// TwinCAT 3 PLC project TC_Robot_Contro_System_Test
// ProgramVersion: 3.1.4020.4
// libraries:
//   Tc2_MC2, * (Beckhoff Automation GmbH)
//   Tc2_Standard, * (Beckhoff Automation GmbH)
//   Tc2_System, * (Beckhoff Automation GmbH)
//   Tc3_Module, * (Beckhoff Automation GmbH)
//   VisuDialogs, * (System)
// project tree:
//   DUTs/Axis/ Axis.TcPOU
//   DUTs/Delay/ Delay.TcPOU (not stored)
//   DUTs/Filter_Current/ E_TcMatSimDataAreaType_1.TcDUT (not stored), FB_Filter_Current_Hexapod_Robot.TcPOU, FB_TcMatSimObject_1.TcPOU (not stored), ST_Filter_Current_Hexapod_Robot_InitData.TcDUT (not stored), ST_Filter_Current_Hexapod_Robot_Input.TcDUT, ST_Filter_Current_Hexapod_Robot_Output.TcDUT (not stored), ST_TcMatSimObjectDataAreaInfo_1.TcDUT (not stored)
//   DUTs/Hexapod_Leg/ Hexapod_Leg.TcPOU (not stored)
//   DUTs/Mapping/ Leg_Control_Mapping_Model.TcPOU (not stored), Leg_Model_Mapping_Control.TcPOU (not stored), Variable_Control_Mapping_Model.TcPOU (not stored), Variable_Model_Mapping_Control.TcPOU (not stored)
//   DUTs/Robot_Simulink/ E_TcMatSimDataAreaType.TcDUT, FB_TcMatSimObject.TcPOU (not stored), FB_Welding_Control_Circle_86s.TcPOU, ST_TcMatSimObjectDataAreaInfo.TcDUT, ST_Welding_Control_Circle_86s_InitData.TcDUT (not stored), ST_Welding_Control_Circle_86s_Input.TcDUT, ST_Welding_Control_Circle_86s_Output.TcDUT
//   / GlobalTextList.TcGTLO (not stored), PlcTask.TcTTO (not stored), Simulink_Test.TcTTO, 视图管理器.TcVMO (not stored)
//   POUs/ MAIN.TcPOU, Simulink_Model_Generator.TcPOU
//   VISUs/ Visu_Home.TcVIS (not stored), Visu_Power.TcVIS, Visu_Reset.TcVIS (not stored), Visu_SimulinkMove.TcVIS (not stored), Visu_Stand.TcVIS (not stored)
// real-time tasks:
//   TASK PlcTask: cycle T#1ms, priority 8, ADS port 350
//   TASK Simulink_Test: cycle T#1ms, priority 10, ADS port 351
// motion (NC):
//   TASK NC-Task 1 SAF: cycle T#1ms, priority 4, ADS port 501
//   TASK NC-Task 1 SVB: cycle T#1ms, priority 6, ADS port 511
//   AXIS Axis 1 (id 1)
//     Velo: SlowManual=10, FastManual=20
//     OtherSettings: AllowMotionCmdToSlave=true
//     encoder EncType=19
//       EncPara: ScaleFactorNumerator=0.000152590218967, MaxCount=#xffffffff
//     drive DrvType=16
//       DrvPara: MaxCount=#xffffffff
//         TimeComp: TaskDelayCycles=1
//     controller CtrType=1
//       CtrPara: PriorControlFactor=1
//         Observer: BandWidth=20
//   AXIS Axis 2 (id 2)
//     Velo: SlowManual=10, FastManual=20
//     OtherSettings: AllowMotionCmdToSlave=true
//     encoder EncType=19
//       EncPara: ScaleFactorNumerator=0.000152590218967, MaxCount=#xffffffff
//     drive DrvType=16
//       DrvPara: MaxCount=#xffffffff
//         TimeComp: TaskDelayCycles=1
//     controller CtrType=1
//       CtrPara: PriorControlFactor=1
//         Observer: BandWidth=20
//   AXIS Axis 3 (id 3)
//     Velo: SlowManual=10, FastManual=20
//     OtherSettings: AllowMotionCmdToSlave=true
//     encoder EncType=19
//       EncPara: ScaleFactorNumerator=0.000152590218967, MaxCount=#xffffffff
//     drive DrvType=16
//       DrvPara: MaxCount=#xffffffff
//         TimeComp: TaskDelayCycles=1
//     controller CtrType=1
//       CtrPara: PriorControlFactor=1
//         Observer: BandWidth=20
//   AXIS Axis 4 (id 4)
//     Velo: SlowManual=10, FastManual=20
//     OtherSettings: AllowMotionCmdToSlave=true
//     encoder EncType=19
//       EncPara: ScaleFactorNumerator=0.000152590218967, MaxCount=#xffffffff
//     drive DrvType=16
//       DrvPara: MaxCount=#xffffffff
//         TimeComp: TaskDelayCycles=1
//     controller CtrType=1
//       CtrPara: PriorControlFactor=1
//         Observer: BandWidth=20
//   AXIS Axis 5 (id 5)
//     Velo: SlowManual=10, FastManual=20
//     OtherSettings: AllowMotionCmdToSlave=true
//     encoder EncType=19
//       EncPara: ScaleFactorNumerator=0.000152590218967, MaxCount=#xffffffff
//     drive DrvType=16
//       DrvPara: MaxCount=#xffffffff
//         TimeComp: TaskDelayCycles=1
//     controller CtrType=1
//       CtrPara: PriorControlFactor=1
//         Observer: BandWidth=20
//   AXIS Axis 6 (id 6)
//     Velo: SlowManual=10, FastManual=20
//     OtherSettings: AllowMotionCmdToSlave=true
//     encoder EncType=19
//       EncPara: ScaleFactorNumerator=0.000152590218967, MaxCount=#xffffffff
//     drive DrvType=16
//       DrvPara: MaxCount=#xffffffff
//         TimeComp: TaskDelayCycles=1
//     controller CtrType=1
//       CtrPara: PriorControlFactor=1
//         Observer: BandWidth=20
//   AXIS Axis 7 (id 7)
//     Velo: SlowManual=10, FastManual=20
//     OtherSettings: AllowMotionCmdToSlave=true
//     encoder EncType=19
//       EncPara: ScaleFactorNumerator=0.000152590218967, MaxCount=#xffffffff
//     drive DrvType=16
//       DrvPara: MaxCount=#xffffffff
//         TimeComp: TaskDelayCycles=1
//     controller CtrType=1
//       CtrPara: PriorControlFactor=1
//         Observer: BandWidth=20
//   AXIS Axis 8 (id 8)
//     Velo: SlowManual=10, FastManual=20
//     OtherSettings: AllowMotionCmdToSlave=true
//     encoder EncType=19
//       EncPara: ScaleFactorNumerator=0.000152590218967, MaxCount=#xffffffff
//     drive DrvType=16
//       DrvPara: MaxCount=#xffffffff
//         TimeComp: TaskDelayCycles=1
//     controller CtrType=1
//       CtrPara: PriorControlFactor=1
//         Observer: BandWidth=20
//   AXIS Axis 9 (id 9)
//     Velo: SlowManual=10, FastManual=20
//     OtherSettings: AllowMotionCmdToSlave=true
//     encoder EncType=19
//       EncPara: ScaleFactorNumerator=0.000152590218967, MaxCount=#xffffffff
//     drive DrvType=16
//       DrvPara: MaxCount=#xffffffff
//         TimeComp: TaskDelayCycles=1
//     controller CtrType=1
//       CtrPara: PriorControlFactor=1
//         Observer: BandWidth=20
//   AXIS Axis 10 (id 10)
//     Velo: SlowManual=10, FastManual=20
//     OtherSettings: AllowMotionCmdToSlave=true
//     encoder EncType=19
//       EncPara: ScaleFactorNumerator=0.000152590218967, MaxCount=#xffffffff
//     drive DrvType=16
//       DrvPara: MaxCount=#xffffffff
//         TimeComp: TaskDelayCycles=1
//     controller CtrType=1
//       CtrPara: PriorControlFactor=1
//         Observer: BandWidth=20
//   AXIS Axis 11 (id 11)
//     Velo: SlowManual=10, FastManual=20
//     OtherSettings: AllowMotionCmdToSlave=true
//     encoder EncType=19
//       EncPara: ScaleFactorNumerator=0.000152590218967, MaxCount=#xffffffff
//     drive DrvType=16
//       DrvPara: MaxCount=#xffffffff
//         TimeComp: TaskDelayCycles=1
//     controller CtrType=1
//       CtrPara: PriorControlFactor=1
//         Observer: BandWidth=20
//   AXIS Axis 12 (id 12)
//     Velo: SlowManual=10, FastManual=20
//     OtherSettings: AllowMotionCmdToSlave=true
//     encoder EncType=19
//       EncPara: ScaleFactorNumerator=0.000152590218967, MaxCount=#xffffffff
//     drive DrvType=16
//       DrvPara: MaxCount=#xffffffff
//         TimeComp: TaskDelayCycles=1
//     controller CtrType=1
//       CtrPara: PriorControlFactor=1
//         Observer: BandWidth=20
//   AXIS Axis 13 (id 13)
//     Velo: SlowManual=10, FastManual=20
//     OtherSettings: AllowMotionCmdToSlave=true
//     encoder EncType=19
//       EncPara: ScaleFactorNumerator=0.000152590218967, MaxCount=#xffffffff
//     drive DrvType=16
//       DrvPara: MaxCount=#xffffffff
//         TimeComp: TaskDelayCycles=1
//     controller CtrType=1
//       CtrPara: PriorControlFactor=1
//         Observer: BandWidth=20
//   AXIS Axis 14 (id 14)
//     Velo: SlowManual=10, FastManual=20
//     OtherSettings: AllowMotionCmdToSlave=true
//     encoder EncType=19
//       EncPara: ScaleFactorNumerator=0.000152590218967, MaxCount=#xffffffff
//     drive DrvType=16
//       DrvPara: MaxCount=#xffffffff
//         TimeComp: TaskDelayCycles=1
//     controller CtrType=1
//       CtrPara: PriorControlFactor=1
//         Observer: BandWidth=20
//   AXIS Axis 15 (id 15)
//     Velo: SlowManual=10, FastManual=20
//     OtherSettings: AllowMotionCmdToSlave=true
//     encoder EncType=19
//       EncPara: ScaleFactorNumerator=0.000152590218967, MaxCount=#xffffffff
//     drive DrvType=16
//       DrvPara: MaxCount=#xffffffff
//         TimeComp: TaskDelayCycles=1
//     controller CtrType=1
//       CtrPara: PriorControlFactor=1
//         Observer: BandWidth=20
//   AXIS Axis 16 (id 16)
//     Velo: SlowManual=10, FastManual=20
//     OtherSettings: AllowMotionCmdToSlave=true
//     encoder EncType=19
//       EncPara: ScaleFactorNumerator=0.000152590218967, MaxCount=#xffffffff
//     drive DrvType=16
//       DrvPara: MaxCount=#xffffffff
//         TimeComp: TaskDelayCycles=1
//     controller CtrType=1
//       CtrPara: PriorControlFactor=1
//         Observer: BandWidth=20
//   AXIS Axis 17 (id 17)
//     Velo: SlowManual=10, FastManual=20
//     OtherSettings: AllowMotionCmdToSlave=true
//     encoder EncType=19
//       EncPara: ScaleFactorNumerator=0.000152590218967, MaxCount=#xffffffff
//     drive DrvType=16
//       DrvPara: MaxCount=#xffffffff
//         TimeComp: TaskDelayCycles=1
//     controller CtrType=1
//       CtrPara: PriorControlFactor=1
//         Observer: BandWidth=20
//   AXIS Axis 18 (id 18)
//     Velo: SlowManual=10, FastManual=20
//     OtherSettings: AllowMotionCmdToSlave=true
//     encoder EncType=19
//       EncPara: ScaleFactorNumerator=0.000152590218967, MaxCount=#xffffffff
//     drive DrvType=16
//       DrvPara: MaxCount=#xffffffff
//         TimeComp: TaskDelayCycles=1
//     controller CtrType=1
//       CtrPara: PriorControlFactor=1
//         Observer: BandWidth=20
// I/O:
//   DEVICE Device 3 (EtherCAT), AmsNetId 5.41.150.106.4.1
//     Drive 1 (Elmo Drive) [Gold EtherCAT GCON Drive Rev:0x000103F6]
//     Drive 2 (Elmo Drive) [Gold EtherCAT GCON Drive Rev:0x000103F6]
//     Drive 3 (Elmo Drive) [Gold EtherCAT GCON Drive Rev:0x000103F6]
//     Drive 4 (Elmo Drive) [Gold EtherCAT GCON Drive Rev:0x000103F6]
//     Drive 5 (Elmo Drive) [Gold EtherCAT GCON Drive Rev:0x000103F6]
//     Drive 6 (Elmo Drive) [Gold EtherCAT GCON Drive Rev:0x000103F6]
//     Drive 7 (Elmo Drive) [Gold EtherCAT GCON Drive Rev:0x000103F6]
//     Drive 8 (Elmo Drive) [Gold EtherCAT GCON Drive Rev:0x000103F6]
//     Drive 9 (Elmo Drive) [Gold EtherCAT GCON Drive Rev:0x000103F6]
//     Drive 10 (Elmo Drive) [Gold EtherCAT GCON Drive Rev:0x000103F6]
//     Drive 11 (Elmo Drive) [Gold EtherCAT GCON Drive Rev:0x000103F6]
//     Drive 12 (Elmo Drive) [Gold EtherCAT GCON Drive Rev:0x000103F6]
//     Drive 13 (Elmo Drive) [Gold EtherCAT GCON Drive Rev:0x000103F6]
//     Drive 14 (Elmo Drive) [Gold EtherCAT GCON Drive Rev:0x000103F6]
//     Drive 15 (Elmo Drive) [Gold EtherCAT GCON Drive Rev:0x000103F6]
//     Drive 16 (Elmo Drive) [Gold EtherCAT GCON Drive Rev:0x000103F6]
//     Drive 17 (Elmo Drive) [Gold EtherCAT GCON Drive Rev:0x000103F6]
//     Drive 18 (Elmo Drive) [Gold EtherCAT GCON Drive Rev:0x000103F6]
// variable links:
//   NC-Task 1 SAF/Axes/Axis 1 <-> Device 3 (EtherCAT)/Drive 1 (Elmo Drive)
//     Drive/Inputs/In/nDcOutputTime <-> InfoData/DcOutputShift
//     Drive/Inputs/In/nState1 <-> Inputs/Status word
//     Drive/Inputs/In/nState2 <-> Inputs/Status word @bit 8
//     Drive/Inputs/In/nState4 @bit 1 <-> WcState/InputToggle
//     Drive/Inputs/In/nState4 <-> WcState/WcState
//     Drive/Outputs/Out/nCtrl1 <-> Outputs/Control word
//     Drive/Outputs/Out/nCtrl2 <-> Outputs/Control word @bit 8
//     Drive/Outputs/Out/nDataOut1 <-> Outputs/Target Position
//     Enc/Inputs/In/nDataIn1 <-> Inputs/Position actual value
//     Enc/Inputs/In/nDcInputTime <-> InfoData/DcInputShift
//     Enc/Inputs/In/nState4 @bit 1 <-> WcState/InputToggle
//     Enc/Inputs/In/nState4 <-> WcState/WcState
//   NC-Task 1 SAF/Axes/Axis 10 <-> Device 3 (EtherCAT)/Drive 10 (Elmo Drive)
//     Drive/Inputs/In/nDcOutputTime <-> InfoData/DcOutputShift
//     Drive/Inputs/In/nState1 <-> Inputs/Status word
//     Drive/Inputs/In/nState2 <-> Inputs/Status word @bit 8
//     Drive/Inputs/In/nState4 @bit 1 <-> WcState/InputToggle
//     Drive/Inputs/In/nState4 <-> WcState/WcState
//     Drive/Outputs/Out/nCtrl1 <-> Outputs/Control word
//     Drive/Outputs/Out/nCtrl2 <-> Outputs/Control word @bit 8
//     Drive/Outputs/Out/nDataOut1 <-> Outputs/Target Position
//     Enc/Inputs/In/nDataIn1 <-> Inputs/Position actual value
//     Enc/Inputs/In/nDcInputTime <-> InfoData/DcInputShift
//     Enc/Inputs/In/nState4 @bit 1 <-> WcState/InputToggle
//     Enc/Inputs/In/nState4 <-> WcState/WcState
//   NC-Task 1 SAF/Axes/Axis 11 <-> Device 3 (EtherCAT)/Drive 11 (Elmo Drive)
//     Drive/Inputs/In/nDcOutputTime <-> InfoData/DcOutputShift
//     Drive/Inputs/In/nState1 <-> Inputs/Status word
//     Drive/Inputs/In/nState2 <-> Inputs/Status word @bit 8
//     Drive/Inputs/In/nState4 @bit 1 <-> WcState/InputToggle
//     Drive/Inputs/In/nState4 <-> WcState/WcState
//     Drive/Outputs/Out/nCtrl1 <-> Outputs/Control word
//     Drive/Outputs/Out/nCtrl2 <-> Outputs/Control word @bit 8
//     Drive/Outputs/Out/nDataOut1 <-> Outputs/Target Position
//     Enc/Inputs/In/nDataIn1 <-> Inputs/Position actual value
//     Enc/Inputs/In/nDcInputTime <-> InfoData/DcInputShift
//     Enc/Inputs/In/nState4 @bit 1 <-> WcState/InputToggle
//     Enc/Inputs/In/nState4 <-> WcState/WcState
//   NC-Task 1 SAF/Axes/Axis 12 <-> Device 3 (EtherCAT)/Drive 12 (Elmo Drive)
//     Drive/Inputs/In/nDcOutputTime <-> InfoData/DcOutputShift
//     Drive/Inputs/In/nState1 <-> Inputs/Status word
//     Drive/Inputs/In/nState2 <-> Inputs/Status word @bit 8
//     Drive/Inputs/In/nState4 @bit 1 <-> WcState/InputToggle
//     Drive/Inputs/In/nState4 <-> WcState/WcState
//     Drive/Outputs/Out/nCtrl1 <-> Outputs/Control word
//     Drive/Outputs/Out/nCtrl2 <-> Outputs/Control word @bit 8
//     Drive/Outputs/Out/nDataOut1 <-> Outputs/Target Position
//     Enc/Inputs/In/nDataIn1 <-> Inputs/Position actual value
//     Enc/Inputs/In/nDcInputTime <-> InfoData/DcInputShift
//     Enc/Inputs/In/nState4 @bit 1 <-> WcState/InputToggle
//     Enc/Inputs/In/nState4 <-> WcState/WcState
//   NC-Task 1 SAF/Axes/Axis 13 <-> Device 3 (EtherCAT)/Drive 13 (Elmo Drive)
//     Drive/Inputs/In/nDcOutputTime <-> InfoData/DcOutputShift
//     Drive/Inputs/In/nState1 <-> Inputs/Status word
//     Drive/Inputs/In/nState2 <-> Inputs/Status word @bit 8
//     Drive/Inputs/In/nState4 @bit 1 <-> WcState/InputToggle
//     Drive/Inputs/In/nState4 <-> WcState/WcState
//     Drive/Outputs/Out/nCtrl1 <-> Outputs/Control word
//     Drive/Outputs/Out/nCtrl2 <-> Outputs/Control word @bit 8
//     Drive/Outputs/Out/nDataOut1 <-> Outputs/Target Position
//     Enc/Inputs/In/nDataIn1 <-> Inputs/Position actual value
//     Enc/Inputs/In/nDcInputTime <-> InfoData/DcInputShift
//     Enc/Inputs/In/nState4 @bit 1 <-> WcState/InputToggle
//     Enc/Inputs/In/nState4 <-> WcState/WcState
//   NC-Task 1 SAF/Axes/Axis 14 <-> Device 3 (EtherCAT)/Drive 14 (Elmo Drive)
//     Drive/Inputs/In/nDcOutputTime <-> InfoData/DcOutputShift
//     Drive/Inputs/In/nState1 <-> Inputs/Status word
//     Drive/Inputs/In/nState2 <-> Inputs/Status word @bit 8
//     Drive/Inputs/In/nState4 @bit 1 <-> WcState/InputToggle
//     Drive/Inputs/In/nState4 <-> WcState/WcState
//     Drive/Outputs/Out/nCtrl1 <-> Outputs/Control word
//     Drive/Outputs/Out/nCtrl2 <-> Outputs/Control word @bit 8
//     Drive/Outputs/Out/nDataOut1 <-> Outputs/Target Position
//     Enc/Inputs/In/nDataIn1 <-> Inputs/Position actual value
//     Enc/Inputs/In/nDcInputTime <-> InfoData/DcInputShift
//     Enc/Inputs/In/nState4 @bit 1 <-> WcState/InputToggle
//     Enc/Inputs/In/nState4 <-> WcState/WcState
//   NC-Task 1 SAF/Axes/Axis 15 <-> Device 3 (EtherCAT)/Drive 15 (Elmo Drive)
//     Drive/Inputs/In/nDcOutputTime <-> InfoData/DcOutputShift
//     Drive/Inputs/In/nState1 <-> Inputs/Status word
//     Drive/Inputs/In/nState2 <-> Inputs/Status word @bit 8
//     Drive/Inputs/In/nState4 @bit 1 <-> WcState/InputToggle
//     Drive/Inputs/In/nState4 <-> WcState/WcState
//     Drive/Outputs/Out/nCtrl1 <-> Outputs/Control word
//     Drive/Outputs/Out/nCtrl2 <-> Outputs/Control word @bit 8
//     Drive/Outputs/Out/nDataOut1 <-> Outputs/Target Position
//     Enc/Inputs/In/nDataIn1 <-> Inputs/Position actual value
//     Enc/Inputs/In/nDcInputTime <-> InfoData/DcInputShift
//     Enc/Inputs/In/nState4 @bit 1 <-> WcState/InputToggle
//     Enc/Inputs/In/nState4 <-> WcState/WcState
//   NC-Task 1 SAF/Axes/Axis 16 <-> Device 3 (EtherCAT)/Drive 16 (Elmo Drive)
//     Drive/Inputs/In/nDcOutputTime <-> InfoData/DcOutputShift
//     Drive/Inputs/In/nState1 <-> Inputs/Status word
//     Drive/Inputs/In/nState2 <-> Inputs/Status word @bit 8
//     Drive/Inputs/In/nState4 @bit 1 <-> WcState/InputToggle
//     Drive/Inputs/In/nState4 <-> WcState/WcState
//     Drive/Outputs/Out/nCtrl1 <-> Outputs/Control word
//     Drive/Outputs/Out/nCtrl2 <-> Outputs/Control word @bit 8
//     Drive/Outputs/Out/nDataOut1 <-> Outputs/Target Position
//     Enc/Inputs/In/nDataIn1 <-> Inputs/Position actual value
//     Enc/Inputs/In/nDcInputTime <-> InfoData/DcInputShift
//     Enc/Inputs/In/nState4 @bit 1 <-> WcState/InputToggle
//     Enc/Inputs/In/nState4 <-> WcState/WcState
//   NC-Task 1 SAF/Axes/Axis 17 <-> Device 3 (EtherCAT)/Drive 17 (Elmo Drive)
//     Drive/Inputs/In/nDcOutputTime <-> InfoData/DcOutputShift
//     Drive/Inputs/In/nState1 <-> Inputs/Status word
//     Drive/Inputs/In/nState2 <-> Inputs/Status word @bit 8
//     Drive/Inputs/In/nState4 @bit 1 <-> WcState/InputToggle
//     Drive/Inputs/In/nState4 <-> WcState/WcState
//     Drive/Outputs/Out/nCtrl1 <-> Outputs/Control word
//     Drive/Outputs/Out/nCtrl2 <-> Outputs/Control word @bit 8
//     Drive/Outputs/Out/nDataOut1 <-> Outputs/Target Position
//     Enc/Inputs/In/nDataIn1 <-> Inputs/Position actual value
//     Enc/Inputs/In/nDcInputTime <-> InfoData/DcInputShift
//     Enc/Inputs/In/nState4 @bit 1 <-> WcState/InputToggle
//     Enc/Inputs/In/nState4 <-> WcState/WcState
//   NC-Task 1 SAF/Axes/Axis 18 <-> Device 3 (EtherCAT)/Drive 18 (Elmo Drive)
//     Drive/Inputs/In/nDcOutputTime <-> InfoData/DcOutputShift
//     Drive/Inputs/In/nState1 <-> Inputs/Status word
//     Drive/Inputs/In/nState2 <-> Inputs/Status word @bit 8
//     Drive/Inputs/In/nState4 @bit 1 <-> WcState/InputToggle
//     Drive/Inputs/In/nState4 <-> WcState/WcState
//     Drive/Outputs/Out/nCtrl1 <-> Outputs/Control word
//     Drive/Outputs/Out/nCtrl2 <-> Outputs/Control word @bit 8
//     Drive/Outputs/Out/nDataOut1 <-> Outputs/Target Position
//     Enc/Inputs/In/nDataIn1 <-> Inputs/Position actual value
//     Enc/Inputs/In/nDcInputTime <-> InfoData/DcInputShift
//     Enc/Inputs/In/nState4 @bit 1 <-> WcState/InputToggle
//     Enc/Inputs/In/nState4 <-> WcState/WcState
//   NC-Task 1 SAF/Axes/Axis 2 <-> Device 3 (EtherCAT)/Drive 2 (Elmo Drive)
//     Drive/Inputs/In/nDcOutputTime <-> InfoData/DcOutputShift
//     Drive/Inputs/In/nState1 <-> Inputs/Status word
//     Drive/Inputs/In/nState2 <-> Inputs/Status word @bit 8
//     Drive/Inputs/In/nState4 @bit 1 <-> WcState/InputToggle
//     Drive/Inputs/In/nState4 <-> WcState/WcState
//     Drive/Outputs/Out/nCtrl1 <-> Outputs/Control word
//     Drive/Outputs/Out/nCtrl2 <-> Outputs/Control word @bit 8
//     Drive/Outputs/Out/nDataOut1 <-> Outputs/Target Position
//     Enc/Inputs/In/nDataIn1 <-> Inputs/Position actual value
//     Enc/Inputs/In/nDcInputTime <-> InfoData/DcInputShift
//     Enc/Inputs/In/nState4 @bit 1 <-> WcState/InputToggle
//     Enc/Inputs/In/nState4 <-> WcState/WcState
//   NC-Task 1 SAF/Axes/Axis 3 <-> Device 3 (EtherCAT)/Drive 3 (Elmo Drive)
//     Drive/Inputs/In/nDcOutputTime <-> InfoData/DcOutputShift
//     Drive/Inputs/In/nState1 <-> Inputs/Status word
//     Drive/Inputs/In/nState2 <-> Inputs/Status word @bit 8
//     Drive/Inputs/In/nState4 @bit 1 <-> WcState/InputToggle
//     Drive/Inputs/In/nState4 <-> WcState/WcState
//     Drive/Outputs/Out/nCtrl1 <-> Outputs/Control word
//     Drive/Outputs/Out/nCtrl2 <-> Outputs/Control word @bit 8
//     Drive/Outputs/Out/nDataOut1 <-> Outputs/Target Position
//     Enc/Inputs/In/nDataIn1 <-> Inputs/Position actual value
//     Enc/Inputs/In/nDcInputTime <-> InfoData/DcInputShift
//     Enc/Inputs/In/nState4 @bit 1 <-> WcState/InputToggle
//     Enc/Inputs/In/nState4 <-> WcState/WcState
//   NC-Task 1 SAF/Axes/Axis 4 <-> Device 3 (EtherCAT)/Drive 4 (Elmo Drive)
//     Drive/Inputs/In/nDcOutputTime <-> InfoData/DcOutputShift
//     Drive/Inputs/In/nState1 <-> Inputs/Status word
//     Drive/Inputs/In/nState2 <-> Inputs/Status word @bit 8
//     Drive/Inputs/In/nState4 @bit 1 <-> WcState/InputToggle
//     Drive/Inputs/In/nState4 <-> WcState/WcState
//     Drive/Outputs/Out/nCtrl1 <-> Outputs/Control word
//     Drive/Outputs/Out/nCtrl2 <-> Outputs/Control word @bit 8
//     Drive/Outputs/Out/nDataOut1 <-> Outputs/Target Position
//     Enc/Inputs/In/nDataIn1 <-> Inputs/Position actual value
//     Enc/Inputs/In/nDcInputTime <-> InfoData/DcInputShift
//     Enc/Inputs/In/nState4 @bit 1 <-> WcState/InputToggle
//     Enc/Inputs/In/nState4 <-> WcState/WcState
//   NC-Task 1 SAF/Axes/Axis 5 <-> Device 3 (EtherCAT)/Drive 5 (Elmo Drive)
//     Drive/Inputs/In/nDcOutputTime <-> InfoData/DcOutputShift
//     Drive/Inputs/In/nState1 <-> Inputs/Status word
//     Drive/Inputs/In/nState2 <-> Inputs/Status word @bit 8
//     Drive/Inputs/In/nState4 @bit 1 <-> WcState/InputToggle
//     Drive/Inputs/In/nState4 <-> WcState/WcState
//     Drive/Outputs/Out/nCtrl1 <-> Outputs/Control word
//     Drive/Outputs/Out/nCtrl2 <-> Outputs/Control word @bit 8
//     Drive/Outputs/Out/nDataOut1 <-> Outputs/Target Position
//     Enc/Inputs/In/nDataIn1 <-> Inputs/Position actual value
//     Enc/Inputs/In/nDcInputTime <-> InfoData/DcInputShift
//     Enc/Inputs/In/nState4 @bit 1 <-> WcState/InputToggle
//     Enc/Inputs/In/nState4 <-> WcState/WcState
//   NC-Task 1 SAF/Axes/Axis 6 <-> Device 3 (EtherCAT)/Drive 6 (Elmo Drive)
//     Drive/Inputs/In/nDcOutputTime <-> InfoData/DcOutputShift
//     Drive/Inputs/In/nState1 <-> Inputs/Status word
//     Drive/Inputs/In/nState2 <-> Inputs/Status word @bit 8
//     Drive/Inputs/In/nState4 @bit 1 <-> WcState/InputToggle
//     Drive/Inputs/In/nState4 <-> WcState/WcState
//     Drive/Outputs/Out/nCtrl1 <-> Outputs/Control word
//     Drive/Outputs/Out/nCtrl2 <-> Outputs/Control word @bit 8
//     Drive/Outputs/Out/nDataOut1 <-> Outputs/Target Position
//     Enc/Inputs/In/nDataIn1 <-> Inputs/Position actual value
//     Enc/Inputs/In/nDcInputTime <-> InfoData/DcInputShift
//     Enc/Inputs/In/nState4 @bit 1 <-> WcState/InputToggle
//     Enc/Inputs/In/nState4 <-> WcState/WcState
//   NC-Task 1 SAF/Axes/Axis 7 <-> Device 3 (EtherCAT)/Drive 7 (Elmo Drive)
//     Drive/Inputs/In/nDcOutputTime <-> InfoData/DcOutputShift
//     Drive/Inputs/In/nState1 <-> Inputs/Status word
//     Drive/Inputs/In/nState2 <-> Inputs/Status word @bit 8
//     Drive/Inputs/In/nState4 @bit 1 <-> WcState/InputToggle
//     Drive/Inputs/In/nState4 <-> WcState/WcState
//     Drive/Outputs/Out/nCtrl1 <-> Outputs/Control word
//     Drive/Outputs/Out/nCtrl2 <-> Outputs/Control word @bit 8
//     Drive/Outputs/Out/nDataOut1 <-> Outputs/Target Position
//     Enc/Inputs/In/nDataIn1 <-> Inputs/Position actual value
//     Enc/Inputs/In/nDcInputTime <-> InfoData/DcInputShift
//     Enc/Inputs/In/nState4 @bit 1 <-> WcState/InputToggle
//     Enc/Inputs/In/nState4 <-> WcState/WcState
//   NC-Task 1 SAF/Axes/Axis 8 <-> Device 3 (EtherCAT)/Drive 8 (Elmo Drive)
//     Drive/Inputs/In/nDcOutputTime <-> InfoData/DcOutputShift
//     Drive/Inputs/In/nState1 <-> Inputs/Status word
//     Drive/Inputs/In/nState2 <-> Inputs/Status word @bit 8
//     Drive/Inputs/In/nState4 @bit 1 <-> WcState/InputToggle
//     Drive/Inputs/In/nState4 <-> WcState/WcState
//     Drive/Outputs/Out/nCtrl1 <-> Outputs/Control word
//     Drive/Outputs/Out/nCtrl2 <-> Outputs/Control word @bit 8
//     Drive/Outputs/Out/nDataOut1 <-> Outputs/Target Position
//     Enc/Inputs/In/nDataIn1 <-> Inputs/Position actual value
//     Enc/Inputs/In/nDcInputTime <-> InfoData/DcInputShift
//     Enc/Inputs/In/nState4 @bit 1 <-> WcState/InputToggle
//     Enc/Inputs/In/nState4 <-> WcState/WcState
//   NC-Task 1 SAF/Axes/Axis 9 <-> Device 3 (EtherCAT)/Drive 9 (Elmo Drive)
//     Drive/Inputs/In/nDcOutputTime <-> InfoData/DcOutputShift
//     Drive/Inputs/In/nState1 <-> Inputs/Status word
//     Drive/Inputs/In/nState2 <-> Inputs/Status word @bit 8
//     Drive/Inputs/In/nState4 @bit 1 <-> WcState/InputToggle
//     Drive/Inputs/In/nState4 <-> WcState/WcState
//     Drive/Outputs/Out/nCtrl1 <-> Outputs/Control word
//     Drive/Outputs/Out/nCtrl2 <-> Outputs/Control word @bit 8
//     Drive/Outputs/Out/nDataOut1 <-> Outputs/Target Position
//     Enc/Inputs/In/nDataIn1 <-> Inputs/Position actual value
//     Enc/Inputs/In/nDcInputTime <-> InfoData/DcInputShift
//     Enc/Inputs/In/nState4 @bit 1 <-> WcState/InputToggle
//     Enc/Inputs/In/nState4 <-> WcState/WcState
//   TC_Robot_Contro_System_Test/TC_Robot_Contro_System_Test Instance <-> Device 3 (EtherCAT)/Drive 1 (Elmo Drive)
//     PlcTask Inputs/MAIN.Current_Turque_Value[1] <-> Inputs_1/Current actual value
//   TC_Robot_Contro_System_Test/TC_Robot_Contro_System_Test Instance <-> Device 3 (EtherCAT)/Drive 10 (Elmo Drive)
//     PlcTask Inputs/MAIN.Current_Turque_Value[10] <-> Inputs_1/Current actual value
//   TC_Robot_Contro_System_Test/TC_Robot_Contro_System_Test Instance <-> Device 3 (EtherCAT)/Drive 11 (Elmo Drive)
//     PlcTask Inputs/MAIN.Current_Turque_Value[11] <-> Inputs_1/Current actual value
//   TC_Robot_Contro_System_Test/TC_Robot_Contro_System_Test Instance <-> Device 3 (EtherCAT)/Drive 12 (Elmo Drive)
//     PlcTask Inputs/MAIN.Current_Turque_Value[12] <-> Inputs_1/Current actual value
//   TC_Robot_Contro_System_Test/TC_Robot_Contro_System_Test Instance <-> Device 3 (EtherCAT)/Drive 13 (Elmo Drive)
//     PlcTask Inputs/MAIN.Current_Turque_Value[13] <-> Inputs_1/Current actual value
//   TC_Robot_Contro_System_Test/TC_Robot_Contro_System_Test Instance <-> Device 3 (EtherCAT)/Drive 14 (Elmo Drive)
//     PlcTask Inputs/MAIN.Current_Turque_Value[14] <-> Inputs_1/Current actual value
//   TC_Robot_Contro_System_Test/TC_Robot_Contro_System_Test Instance <-> Device 3 (EtherCAT)/Drive 15 (Elmo Drive)
//     PlcTask Inputs/MAIN.Current_Turque_Value[15] <-> Inputs_1/Current actual value
//   TC_Robot_Contro_System_Test/TC_Robot_Contro_System_Test Instance <-> Device 3 (EtherCAT)/Drive 16 (Elmo Drive)
//     PlcTask Inputs/MAIN.Current_Turque_Value[16] <-> Inputs_1/Current actual value
//   TC_Robot_Contro_System_Test/TC_Robot_Contro_System_Test Instance <-> Device 3 (EtherCAT)/Drive 17 (Elmo Drive)
//     PlcTask Inputs/MAIN.Current_Turque_Value[17] <-> Inputs_1/Current actual value
//   TC_Robot_Contro_System_Test/TC_Robot_Contro_System_Test Instance <-> Device 3 (EtherCAT)/Drive 18 (Elmo Drive)
//     PlcTask Inputs/MAIN.Current_Turque_Value[18] <-> Inputs_1/Current actual value
//   TC_Robot_Contro_System_Test/TC_Robot_Contro_System_Test Instance <-> Device 3 (EtherCAT)/Drive 2 (Elmo Drive)
//     PlcTask Inputs/MAIN.Current_Turque_Value[2] <-> Inputs_1/Current actual value
//   TC_Robot_Contro_System_Test/TC_Robot_Contro_System_Test Instance <-> Device 3 (EtherCAT)/Drive 3 (Elmo Drive)
//     PlcTask Inputs/MAIN.Current_Turque_Value[3] <-> Inputs_1/Current actual value
//   TC_Robot_Contro_System_Test/TC_Robot_Contro_System_Test Instance <-> Device 3 (EtherCAT)/Drive 4 (Elmo Drive)
//     PlcTask Inputs/MAIN.Current_Turque_Value[4] <-> Inputs_1/Current actual value
//   TC_Robot_Contro_System_Test/TC_Robot_Contro_System_Test Instance <-> Device 3 (EtherCAT)/Drive 5 (Elmo Drive)
//     PlcTask Inputs/MAIN.Current_Turque_Value[5] <-> Inputs_1/Current actual value
//   TC_Robot_Contro_System_Test/TC_Robot_Contro_System_Test Instance <-> Device 3 (EtherCAT)/Drive 6 (Elmo Drive)
//     PlcTask Inputs/MAIN.Current_Turque_Value[6] <-> Inputs_1/Current actual value
//   TC_Robot_Contro_System_Test/TC_Robot_Contro_System_Test Instance <-> Device 3 (EtherCAT)/Drive 7 (Elmo Drive)
//     PlcTask Inputs/MAIN.Current_Turque_Value[7] <-> Inputs_1/Current actual value
//   TC_Robot_Contro_System_Test/TC_Robot_Contro_System_Test Instance <-> Device 3 (EtherCAT)/Drive 8 (Elmo Drive)
//     PlcTask Inputs/MAIN.Current_Turque_Value[8] <-> Inputs_1/Current actual value
//   TC_Robot_Contro_System_Test/TC_Robot_Contro_System_Test Instance <-> Device 3 (EtherCAT)/Drive 9 (Elmo Drive)
//     PlcTask Inputs/MAIN.Current_Turque_Value[9] <-> Inputs_1/Current actual value
//   TC_Robot_Contro_System_Test/TC_Robot_Contro_System_Test Instance <-> NC-Task 1 SAF/Axes/Axis 1
//     PlcTask Inputs/MAIN.Axis_Robot[1].AxisRef.NcToPlc <-> Outputs/ToPlc
//     PlcTask Outputs/MAIN.Axis_Robot[1].AxisRef.PlcToNc <-> Inputs/FromPlc
//   TC_Robot_Contro_System_Test/TC_Robot_Contro_System_Test Instance <-> NC-Task 1 SAF/Axes/Axis 10
//     PlcTask Inputs/MAIN.Axis_Robot[10].AxisRef.NcToPlc <-> Outputs/ToPlc
//     PlcTask Outputs/MAIN.Axis_Robot[10].AxisRef.PlcToNc <-> Inputs/FromPlc
//   TC_Robot_Contro_System_Test/TC_Robot_Contro_System_Test Instance <-> NC-Task 1 SAF/Axes/Axis 11
//     PlcTask Inputs/MAIN.Axis_Robot[11].AxisRef.NcToPlc <-> Outputs/ToPlc
//     PlcTask Outputs/MAIN.Axis_Robot[11].AxisRef.PlcToNc <-> Inputs/FromPlc
//   TC_Robot_Contro_System_Test/TC_Robot_Contro_System_Test Instance <-> NC-Task 1 SAF/Axes/Axis 12
//     PlcTask Inputs/MAIN.Axis_Robot[12].AxisRef.NcToPlc <-> Outputs/ToPlc
//     PlcTask Outputs/MAIN.Axis_Robot[12].AxisRef.PlcToNc <-> Inputs/FromPlc
//   TC_Robot_Contro_System_Test/TC_Robot_Contro_System_Test Instance <-> NC-Task 1 SAF/Axes/Axis 13
//     PlcTask Inputs/MAIN.Axis_Robot[13].AxisRef.NcToPlc <-> Outputs/ToPlc
//     PlcTask Outputs/MAIN.Axis_Robot[13].AxisRef.PlcToNc <-> Inputs/FromPlc
//   TC_Robot_Contro_System_Test/TC_Robot_Contro_System_Test Instance <-> NC-Task 1 SAF/Axes/Axis 14
//     PlcTask Inputs/MAIN.Axis_Robot[14].AxisRef.NcToPlc <-> Outputs/ToPlc
//     PlcTask Outputs/MAIN.Axis_Robot[14].AxisRef.PlcToNc <-> Inputs/FromPlc
//   TC_Robot_Contro_System_Test/TC_Robot_Contro_System_Test Instance <-> NC-Task 1 SAF/Axes/Axis 15
//     PlcTask Inputs/MAIN.Axis_Robot[15].AxisRef.NcToPlc <-> Outputs/ToPlc
//     PlcTask Outputs/MAIN.Axis_Robot[15].AxisRef.PlcToNc <-> Inputs/FromPlc
//   TC_Robot_Contro_System_Test/TC_Robot_Contro_System_Test Instance <-> NC-Task 1 SAF/Axes/Axis 16
//     PlcTask Inputs/MAIN.Axis_Robot[16].AxisRef.NcToPlc <-> Outputs/ToPlc
//     PlcTask Outputs/MAIN.Axis_Robot[16].AxisRef.PlcToNc <-> Inputs/FromPlc
//   TC_Robot_Contro_System_Test/TC_Robot_Contro_System_Test Instance <-> NC-Task 1 SAF/Axes/Axis 17
//     PlcTask Inputs/MAIN.Axis_Robot[17].AxisRef.NcToPlc <-> Outputs/ToPlc
//     PlcTask Outputs/MAIN.Axis_Robot[17].AxisRef.PlcToNc <-> Inputs/FromPlc
//   TC_Robot_Contro_System_Test/TC_Robot_Contro_System_Test Instance <-> NC-Task 1 SAF/Axes/Axis 18
//     PlcTask Inputs/MAIN.Axis_Robot[18].AxisRef.NcToPlc <-> Outputs/ToPlc
//     PlcTask Outputs/MAIN.Axis_Robot[18].AxisRef.PlcToNc <-> Inputs/FromPlc
//   TC_Robot_Contro_System_Test/TC_Robot_Contro_System_Test Instance <-> NC-Task 1 SAF/Axes/Axis 2
//     PlcTask Inputs/MAIN.Axis_Robot[2].AxisRef.NcToPlc <-> Outputs/ToPlc
//     PlcTask Outputs/MAIN.Axis_Robot[2].AxisRef.PlcToNc <-> Inputs/FromPlc
//   TC_Robot_Contro_System_Test/TC_Robot_Contro_System_Test Instance <-> NC-Task 1 SAF/Axes/Axis 3
//     PlcTask Inputs/MAIN.Axis_Robot[3].AxisRef.NcToPlc <-> Outputs/ToPlc
//     PlcTask Outputs/MAIN.Axis_Robot[3].AxisRef.PlcToNc <-> Inputs/FromPlc
//   TC_Robot_Contro_System_Test/TC_Robot_Contro_System_Test Instance <-> NC-Task 1 SAF/Axes/Axis 4
//     PlcTask Inputs/MAIN.Axis_Robot[4].AxisRef.NcToPlc <-> Outputs/ToPlc
//     PlcTask Outputs/MAIN.Axis_Robot[4].AxisRef.PlcToNc <-> Inputs/FromPlc
//   TC_Robot_Contro_System_Test/TC_Robot_Contro_System_Test Instance <-> NC-Task 1 SAF/Axes/Axis 5
//     PlcTask Inputs/MAIN.Axis_Robot[5].AxisRef.NcToPlc <-> Outputs/ToPlc
//     PlcTask Outputs/MAIN.Axis_Robot[5].AxisRef.PlcToNc <-> Inputs/FromPlc
//   TC_Robot_Contro_System_Test/TC_Robot_Contro_System_Test Instance <-> NC-Task 1 SAF/Axes/Axis 6
//     PlcTask Inputs/MAIN.Axis_Robot[6].AxisRef.NcToPlc <-> Outputs/ToPlc
//     PlcTask Outputs/MAIN.Axis_Robot[6].AxisRef.PlcToNc <-> Inputs/FromPlc
//   TC_Robot_Contro_System_Test/TC_Robot_Contro_System_Test Instance <-> NC-Task 1 SAF/Axes/Axis 7
//     PlcTask Inputs/MAIN.Axis_Robot[7].AxisRef.NcToPlc <-> Outputs/ToPlc
//     PlcTask Outputs/MAIN.Axis_Robot[7].AxisRef.PlcToNc <-> Inputs/FromPlc
//   TC_Robot_Contro_System_Test/TC_Robot_Contro_System_Test Instance <-> NC-Task 1 SAF/Axes/Axis 8
//     PlcTask Inputs/MAIN.Axis_Robot[8].AxisRef.NcToPlc <-> Outputs/ToPlc
//     PlcTask Outputs/MAIN.Axis_Robot[8].AxisRef.PlcToNc <-> Inputs/FromPlc
//   TC_Robot_Contro_System_Test/TC_Robot_Contro_System_Test Instance <-> NC-Task 1 SAF/Axes/Axis 9
//     PlcTask Inputs/MAIN.Axis_Robot[9].AxisRef.NcToPlc <-> Outputs/ToPlc
//     PlcTask Outputs/MAIN.Axis_Robot[9].AxisRef.PlcToNc <-> Inputs/FromPlc

CONFIGURATION TC_Robot_Contro_System_Test
    RESOURCE PLC ON TwinCAT3
        TASK Simulink_Test(INTERVAL := T#1ms, PRIORITY := 10);
        PROGRAM Simulink_Model_Generator WITH Simulink_Test : Simulink_Model_Generator;
    END_RESOURCE
END_CONFIGURATION

// ---- DUTs/Filter_Current/ST_Filter_Current_Hexapod_Robot_Input.TcDUT
TYPE ST_Filter_Current_Hexapod_Robot_Input :
STRUCT
	Current_Motor: matrix_18_real_T;
END_STRUCT
END_TYPE

// ---- DUTs/Robot_Simulink/E_TcMatSimDataAreaType.TcDUT
TYPE E_TcMatSimDataAreaType :
(
	NotSpecified := 0,
	Standard,
	InputSrc,
	InputDst,
	OutputSrc,
	OutputDst,
	InternalDa,
	MArea,
	RetainDa
);
END_TYPE

// ---- DUTs/Robot_Simulink/ST_TcMatSimObjectDataAreaInfo.TcDUT
TYPE ST_TcMatSimObjectDataAreaInfo :
STRUCT
	pPlcVar: PVOID;
	pModuleProcImg: PVOID;
	nSize: UDINT;
	nDataAreaId: UDINT;
	eDataAreaType: E_TcMatSimDataAreaType;
END_STRUCT
END_TYPE

// ---- DUTs/Robot_Simulink/ST_Welding_Control_Circle_86s_Input.TcDUT
TYPE ST_Welding_Control_Circle_86s_Input :
STRUCT
	t: LREAL;
END_STRUCT
END_TYPE

// ---- DUTs/Robot_Simulink/ST_Welding_Control_Circle_86s_Output.TcDUT
TYPE ST_Welding_Control_Circle_86s_Output :
STRUCT
	Disp_P: matrix_18_real_T;
END_STRUCT
END_TYPE

// ---- POUs/Simulink_Model_Generator.TcPOU
PROGRAM Simulink_Model_Generator
VAR_INPUT
	
	Axis_Number 		: INT;							// 定义轴数目
	
	ExSetPoint_Execute	: BOOL;							// 机器人外部信号发生使能
	ExtSetPointEnable	: BOOL;							// 外部信号发生信号
	ExtSetPointDisable	: BOOL;							// 外部信号结束信号
	
	T_ALL				: LREAL:=100;						// Simulink模型运动总时长
	t_Interval			: LREAL:=0.001;						// 取样时间间隔，默认为1ms
	t					: LREAL:=0;							// 取样当前时间变量，以0为起点
	
	// ====================Simulink模块相关=====================
	Robot_Simulink		: FB_Welding_Control_Circle_86s(oid:=16#01010020);	// Simulink模型定义
	Mapping_Position	: Variable_Model_Mapping_Control;	// 变量映射			
	
	Filter_Current  	: FB_Filter_Current_Hexapod_Robot(oid:=16#01010030);
	Mapping_Current_Filter	: Variable_Control_Mapping_Model;		// 变量映射	

	
END_VAR
VAR
	Leg_Number			: INT;							// 定义机器人腿数
END_VAR
VAR_OUTPUT
	Model_Position		: ARRAY[1..18] OF LREAL;			// Simulink中各个腿的位置
	ExSetPoint_Position	: ARRAY[1..18] OF LREAL;			// 外部信号位置
	
	Current_Turque_Filter  	: ARRAY[1..18] OF LREAL;		// 滤波后电流
	Current_Turque_Leg		: ARRAY[1..18] OF LREAL;		// Mapping后的电流
	Difference_Position	: ARRAY[1..18] OF LREAL;			// 实际位置与输入位置差值
END_VAR

// =======================子程序使能(永久运行)===================
Variable_Monitor();			// 变量监测子程序使能
Logic_Control();			// 逻辑控制子程序使能
Variable_Set();				// 各动作速度子程序使能

// =======================模型使能=======================
IF ExSetPoint_Execute OR MAIN.Home_Execute THEN
	Robot_Simulink.Execute();	// Simulink模型使能
END_IF

IF MAIN.Power_Execute THEN
	Filter_Current.Execute();
END_IF

// =======================外部信号运动程序=======================
IF ExSetPoint_Execute THEN
	//SetGenerator();			// 使能外部信号发生子程序
	FOR Axis_Number := 1 TO 18 {BY 1} DO
		MAIN.Axis_Robot[Axis_Number].ExtSetPoint(	Drive_ExtSetPointEnable:= ExtSetPointEnable, 
													Drive_ExtSetPointDisable:= ExtSetPointDisable, 
													ExSetPosition:= ExSetPoint_Position[Axis_Number]);
	END_FOR
END_IF


// ======================外部信号发生=========================
IF ExtSetPointEnable THEN	
	t := t + t_Interval;
	ExtSetPointDisable := FALSE;
END_IF

IF t>=T_ALL THEN
	ExtSetPointEnable := FALSE;
	t:=0;
	ExtSetPointDisable := TRUE;
END_IF

ACTION Leg_Action:
// ===================机器人触地信号转换====================
//IF ExtSetPointEnable THEN
//	FOR Leg_Number := 1 TO 6 {BY 1} DO
//		IF Leg_Home_Set[Leg_Number] THEN		// 在可视化中，Leg_Home_Set为点动
//			Axis_Home_Set[1+(Leg_Number-1)*3] := Leg_Home_Set[Leg_Number];
//			Axis_Home_Set[2+(Leg_Number-1)*3] := Leg_Home_Set[Leg_Number];
//			Axis_Home_Set[3+(Leg_Number-1)*3] := Leg_Home_Set[Leg_Number];
//		ELSIF Home_Done[1+(Leg_Number-1)*3] AND Home_Done[2+(Leg_Number-1)*3] AND Home_Done[3+(Leg_Number-1)*3] THEN
//			Leg_Home_Set[Leg_Number] := FALSE; 
//		END_IF
//	END_FOR
//END_IF
END_ACTION

ACTION Logic_Control:
// =====================外部信号发生逻辑========================
IF ExSetPoint_Execute THEN
	MAIN.Home_Execute := FALSE;						// 外部信号发生使能时，机器人调零必须结束
	MAIN.Move_Execute :=0;							// 外部信号发生时，不能进行其他运动
ELSIF NOT ExSetPoint_Execute THEN
	ExtSetPointEnable := 0;						// 外部信号发生不使能时，外部信号不能进入程序
	ExtSetPointDisable :=0;
ELSIF ExtSetPointDisable THEN
	ExtSetPointEnable :=0;						// 外部信号发生停止与外部信号发生开始不能同时进行
END_IF

IF MAIN.Home_Execute OR MAIN.Move_Execute THEN
	ExSetPoint_Execute := FALSE;
END_IF
END_ACTION

ACTION Variable_Monitor:
// ==============实际运动位移和输入位移差值检测区==============
FOR Axis_Number := 1 TO 18 {BY 1} DO
	Difference_Position[Axis_Number] := MAIN.Axis_ActPostion[Axis_Number]- Mapping_Position.Controller_Leg_Variable[Axis_Number]; 
END_FOR

// ===================电流滤波环节===================
FOR Axis_Number := 1 TO 18 {BY 1} DO
	Filter_Current.stInput.Current_Motor[Axis_Number-1] := MAIN.Current_Turque_Value[Axis_Number];
END_FOR	

Current_Turque_Filter := Filter_Current.stOutput.Current_Monitor;
Mapping_Current_Filter(Controller_Leg_Variable:= Current_Turque_Filter, Model_Leg_Variable=> Current_Turque_Leg);
END_ACTION

ACTION Variable_Set:
// ===================外部信号发生电机位置输入值================
FOR Axis_Number := 1 TO 18 {BY 1} DO
	ExSetPoint_Position[Axis_Number]:= Mapping_Position.Controller_Leg_Variable[Axis_Number];
END_FOR

// ===================程序与模型的变量链接===================
Mapping_Position(Model_Leg_Variable:= Model_Position);		// 映射运动学模型中腿编号和控制模型中的电机编号
Robot_Simulink.stInput.t := t;								// 采样时间t与Simulink模型中的采样时间链接
Model_Position := Robot_Simulink.stOutput.Disp_P;			// Simulink中的电机输出位移输入到控制模型
END_ACTION

END_PROGRAM

// ---- DUTs/Robot_Simulink/FB_Welding_Control_Circle_86s.TcPOU
{attribute 'TcDependOnClassFactory' := 'Welding_Control_Circle_86s'}
FUNCTION_BLOCK FB_Welding_Control_Circle_86s EXTENDS FB_TcMatSimObject
VAR_INPUT
	stInput: ST_Welding_Control_Circle_86s_Input;
END_VAR
VAR_OUTPUT
	stOutput: ST_Welding_Control_Circle_86s_Output;
END_VAR
VAR
	stInitData: ST_Welding_Control_Circle_86s_InitData;
	arrDataAreas: ARRAY[1..2] OF ST_TcMatSimObjectDataAreaInfo;
	bParametersVerified: BOOL;
END_VAR

PROPERTY CallBy_Online : TctModuleCallByType
GET
hResult := GetObjPara(16#00000000,sizeof(CallBy_Online),adr(CallBy_Online));
END_GET
SET
hResult := SetObjPara(16#00000000,sizeof(CallBy_Online),adr(CallBy_Online));
END_SET
END_PROPERTY

PROPERTY CallBy_Startup : TctModuleCallByType
GET
CallBy_Startup := stInitData.CallBy;
END_GET
SET
stInitData.CallBy := CallBy_Startup;
END_SET
END_PROPERTY

PROPERTY ContextInfoArr_0_TaskCycleTimeNs_Online : UDINT
GET
hResult := GetObjPara(16#03002080,sizeof(ContextInfoArr_0_TaskCycleTimeNs_Online),adr(ContextInfoArr_0_TaskCycleTimeNs_Online));
END_GET
SET
hResult := SetObjPara(16#03002080,sizeof(ContextInfoArr_0_TaskCycleTimeNs_Online),adr(ContextInfoArr_0_TaskCycleTimeNs_Online));
END_SET
END_PROPERTY

PROPERTY ContextInfoArr_0_TaskCycleTimeNs_Startup : UDINT
GET
ContextInfoArr_0_TaskCycleTimeNs_Startup := stInitData.ContextInfoArr_0_TaskCycleTimeNs;
END_GET
SET
stInitData.ContextInfoArr_0_TaskCycleTimeNs := ContextInfoArr_0_TaskCycleTimeNs_Startup;
END_SET
END_PROPERTY

PROPERTY ContextInfoArr_0_TaskOid_Online : OTCID
GET
hResult := GetObjPara(16#03002060,sizeof(ContextInfoArr_0_TaskOid_Online),adr(ContextInfoArr_0_TaskOid_Online));
END_GET
SET
hResult := SetObjPara(16#03002060,sizeof(ContextInfoArr_0_TaskOid_Online),adr(ContextInfoArr_0_TaskOid_Online));
END_SET
END_PROPERTY

PROPERTY ContextInfoArr_0_TaskOid_Startup : OTCID
GET
ContextInfoArr_0_TaskOid_Startup := stInitData.ContextInfoArr_0_TaskOid;
END_GET
SET
stInitData.ContextInfoArr_0_TaskOid := ContextInfoArr_0_TaskOid_Startup;
END_SET
END_PROPERTY

PROPERTY ContextInfoArr_0_TaskPort_Online : UINT
GET
hResult := GetObjPara(16#03002090,sizeof(ContextInfoArr_0_TaskPort_Online),adr(ContextInfoArr_0_TaskPort_Online));
END_GET
SET
hResult := SetObjPara(16#03002090,sizeof(ContextInfoArr_0_TaskPort_Online),adr(ContextInfoArr_0_TaskPort_Online));
END_SET
END_PROPERTY

PROPERTY ContextInfoArr_0_TaskPort_Startup : UINT
GET
ContextInfoArr_0_TaskPort_Startup := stInitData.ContextInfoArr_0_TaskPort;
END_GET
SET
stInitData.ContextInfoArr_0_TaskPort := ContextInfoArr_0_TaskPort_Startup;
END_SET
END_PROPERTY

PROPERTY ContextInfoArr_0_TaskPriority_Online : UDINT
GET
hResult := GetObjPara(16#03002070,sizeof(ContextInfoArr_0_TaskPriority_Online),adr(ContextInfoArr_0_TaskPriority_Online));
END_GET
SET
hResult := SetObjPara(16#03002070,sizeof(ContextInfoArr_0_TaskPriority_Online),adr(ContextInfoArr_0_TaskPriority_Online));
END_SET
END_PROPERTY

PROPERTY ContextInfoArr_0_TaskPriority_Startup : UDINT
GET
ContextInfoArr_0_TaskPriority_Startup := stInitData.ContextInfoArr_0_TaskPriority;
END_GET
SET
stInitData.ContextInfoArr_0_TaskPriority := ContextInfoArr_0_TaskPriority_Startup;
END_SET
END_PROPERTY

PROPERTY ContextInfoArr_0_TaskSortOrder_Online : UDINT
GET
hResult := GetObjPara(16#030020b0,sizeof(ContextInfoArr_0_TaskSortOrder_Online),adr(ContextInfoArr_0_TaskSortOrder_Online));
END_GET
SET
hResult := SetObjPara(16#030020b0,sizeof(ContextInfoArr_0_TaskSortOrder_Online),adr(ContextInfoArr_0_TaskSortOrder_Online));
END_SET
END_PROPERTY

PROPERTY ContextInfoArr_0_TaskSortOrder_Startup : UDINT
GET
ContextInfoArr_0_TaskSortOrder_Startup := stInitData.ContextInfoArr_0_TaskSortOrder;
END_GET
SET
stInitData.ContextInfoArr_0_TaskSortOrder := ContextInfoArr_0_TaskSortOrder_Startup;
END_SET
END_PROPERTY

PROPERTY CycleUpdateExecuted_Online : BOOL
GET
hResult := GetObjPara(16#00000004,sizeof(CycleUpdateExecuted_Online),adr(CycleUpdateExecuted_Online));
END_GET
SET
hResult := SetObjPara(16#00000004,sizeof(CycleUpdateExecuted_Online),adr(CycleUpdateExecuted_Online));
END_SET
END_PROPERTY

METHOD Execute : HRESULT

IF (SUCCEEDED(hResult)) THEN
  hResult := VerifyParameters();
END_IF

	// update DataArea information
SetDataAreaInfo(ADR(arrDataAreas),2);
	
	// call base method
Execute := SUPER^.Execute();
END_METHOD

PROPERTY ExecuteModelCode_Online : BOOL
GET
hResult := GetObjPara(16#00000008,sizeof(ExecuteModelCode_Online),adr(ExecuteModelCode_Online));
END_GET
SET
hResult := SetObjPara(16#00000008,sizeof(ExecuteModelCode_Online),adr(ExecuteModelCode_Online));
END_SET
END_PROPERTY

PROPERTY ExecuteModelCode_Startup : BOOL
GET
ExecuteModelCode_Startup := stInitData.ExecuteModelCode;
END_GET
SET
stInitData.ExecuteModelCode := ExecuteModelCode_Startup;
END_SET
END_PROPERTY

PROPERTY ExecutionSequence_Online : TctModuleExecutionSequenceType
GET
hResult := GetObjPara(16#00000001,sizeof(ExecutionSequence_Online),adr(ExecutionSequence_Online));
END_GET
SET
hResult := SetObjPara(16#00000001,sizeof(ExecutionSequence_Online),adr(ExecutionSequence_Online));
END_SET
END_PROPERTY

PROPERTY ExecutionSequence_Startup : TctModuleExecutionSequenceType
GET
ExecutionSequence_Startup := stInitData.ExecutionSequence;
END_GET
SET
stInitData.ExecutionSequence := ExecutionSequence_Startup;
END_SET
END_PROPERTY

METHOD FB_init : BOOL
VAR_INPUT
	/// if TRUE, the retain variables are initialized (warm start / cold start)
	bInitRetains: BOOL;
	/// if TRUE, the instance afterwards gets moved into the copy code (online change)
	bInCopyCode: BOOL;
	oid: OTCID;
END_VAR
VAR
	clsId: CLSID;
END_VAR

// initialize flags
bParametersVerified := false;
                    
// set module class id for compatibility check
clsId.Data1 := 16#4f7c9520;
clsId.Data2 := 16#5e7b;
clsId.Data3 := 16#4579;
clsId.Data4[0] := 16#be;
clsId.Data4[1] := 16#6e;
clsId.Data4[2] := 16#10;
clsId.Data4[3] := 16#c0;
clsId.Data4[4] := 16#eb;
clsId.Data4[5] := 16#37;
clsId.Data4[6] := 16#31;
clsId.Data4[7] := 16#6d;

AssignClassId(clsId);
                    
// initialize InitData structure with default values              
stInitData.CallByHdr.indexGroup := 0;
stInitData.CallByHdr.indexOffset := 16#00000000;
stInitData.CallByHdr.cbData := SIZEOF(stInitData.CallBy);
stInitData.CallBy := TctModuleCallByType.Module;
stInitData.ExecutionSequenceHdr.indexGroup := 0;
stInitData.ExecutionSequenceHdr.indexOffset := 16#00000001;
stInitData.ExecutionSequenceHdr.cbData := SIZEOF(stInitData.ExecutionSequence);
stInitData.ExecutionSequence := TctModuleExecutionSequenceType.StateUpdateAfterOutputMapping;
stInitData.StepSizeHdr.indexGroup := 0;
stInitData.StepSizeHdr.indexOffset := 16#00000002;
stInitData.StepSizeHdr.cbData := SIZEOF(stInitData.StepSize);
stInitData.StepSize := TctStepSizeType.UseTaskCycleTime;
stInitData.ExecuteModelCodeHdr.indexGroup := 0;
stInitData.ExecuteModelCodeHdr.indexOffset := 16#00000008;
stInitData.ExecuteModelCodeHdr.cbData := SIZEOF(stInitData.ExecuteModelCode);
stInitData.ExecuteModelCode := 1;
stInitData.ContextInfoArr_0_TaskOidHdr.indexGroup := 0;
stInitData.ContextInfoArr_0_TaskOidHdr.indexOffset := 16#03002060;
stInitData.ContextInfoArr_0_TaskOidHdr.cbData := SIZEOF(stInitData.ContextInfoArr_0_TaskOid);
stInitData.ContextInfoArr_0_TaskPriorityHdr.indexGroup := 0;
stInitData.ContextInfoArr_0_TaskPriorityHdr.indexOffset := 16#03002070;
stInitData.ContextInfoArr_0_TaskPriorityHdr.cbData := SIZEOF(stInitData.ContextInfoArr_0_TaskPriority);
stInitData.ContextInfoArr_0_TaskCycleTimeNsHdr.indexGroup := 0;
stInitData.ContextInfoArr_0_TaskCycleTimeNsHdr.indexOffset := 16#03002080;
stInitData.ContextInfoArr_0_TaskCycleTimeNsHdr.cbData := SIZEOF(stInitData.ContextInfoArr_0_TaskCycleTimeNs);
stInitData.ContextInfoArr_0_TaskPortHdr.indexGroup := 0;
stInitData.ContextInfoArr_0_TaskPortHdr.indexOffset := 16#03002090;
stInitData.ContextInfoArr_0_TaskPortHdr.cbData := SIZEOF(stInitData.ContextInfoArr_0_TaskPort);
stInitData.ContextInfoArr_0_TaskSortOrderHdr.indexGroup := 0;
stInitData.ContextInfoArr_0_TaskSortOrderHdr.indexOffset := 16#030020b0;
stInitData.ContextInfoArr_0_TaskSortOrderHdr.cbData := SIZEOF(stInitData.ContextInfoArr_0_TaskSortOrder);
stInitData.Header.cbData := SIZEOF(stInitData)-SIZEOF(stInitData.Header);
stInitData.Header.uiElmCnt := 9;


// set pointer to InitData structure
SetInitDataInfo(ADR(stInitData));

// set DataArea information
SetDataAreaInfo(ADR(arrDataAreas),2);
arrDataAreas[1].nDataAreaId := 0;
arrDataAreas[1].nSize := SIZEOF(stInput);
arrDataAreas[1].pPlcVar := ADR(stInput);
arrDataAreas[1].pModuleProcImg := 0;
arrDataAreas[1].eDataAreaType := E_TcMatSimDataAreaType.InputDst;
arrDataAreas[2].nDataAreaId := 1;
arrDataAreas[2].nSize := SIZEOF(stOutput);
arrDataAreas[2].pPlcVar := ADR(stOutput);
arrDataAreas[2].pModuleProcImg := 0;
arrDataAreas[2].eDataAreaType := E_TcMatSimDataAreaType.OutputSrc;


// initialize basic interface pointers and return
FB_init := SUCCEEDED(Init(oid));
END_METHOD

PROPERTY InitData : ST_Welding_Control_Circle_86s_InitData
GET
InitData := stInitData;
END_GET
SET
stInitData := InitData;
END_SET
END_PROPERTY

PROPERTY Input_Online : ExtU_output_WeldingDiameter10_T
GET
hResult := GetObjPara(16#80000000,sizeof(Input_Online),adr(Input_Online));
END_GET
SET
hResult := SetObjPara(16#80000000,sizeof(Input_Online),adr(Input_Online));
END_SET
END_PROPERTY

{attribute 'object_name' := 'Internal_SetObjState'}
METHOD PROTECTED Internal_SetObjState
VAR_INPUT
	hr: REFERENCE TO HRESULT;
	nextState: TCOM_STATE;
END_VAR

// update pointer to InitData structure
SetInitDataInfo(ADR(stInitData));
// call base method
SUPER^.Internal_SetObjState(hr,nextState);
END_METHOD

PROPERTY MdlInitialized_Online : BOOL
GET
hResult := GetObjPara(16#00000003,sizeof(MdlInitialized_Online),adr(MdlInitialized_Online));
END_GET
SET
hResult := SetObjPara(16#00000003,sizeof(MdlInitialized_Online),adr(MdlInitialized_Online));
END_SET
END_PROPERTY

PROPERTY ModuleBuildInfo_Online : TctModuleBuildInfoType
GET
hResult := GetObjPara(16#00000007,sizeof(ModuleBuildInfo_Online),adr(ModuleBuildInfo_Online));
END_GET
SET
hResult := SetObjPara(16#00000007,sizeof(ModuleBuildInfo_Online),adr(ModuleBuildInfo_Online));
END_SET
END_PROPERTY

PROPERTY ModuleInfo_Online : TctModuleInfoType
GET
hResult := GetObjPara(16#00000006,sizeof(ModuleInfo_Online),adr(ModuleInfo_Online));
END_GET
SET
hResult := SetObjPara(16#00000006,sizeof(ModuleInfo_Online),adr(ModuleInfo_Online));
END_SET
END_PROPERTY

{attribute 'object_name' := 'SaveOnlineParametersForInit'}
METHOD SaveOnlineParametersForInit : HRESULT
VAR
	idx: UINT;
	pInitElemHdr: POINTER TO TComInitDataElmHdr;
	pData: PVOID;
	nData: UDINT;
END_VAR
VAR CONSTANT
	nInitDataAlignment: UDINT := 4;
END_VAR

// update pointer to InitData structure
SetInitDataInfo(ADR(stInitData));
// call base method
SaveOnlineParametersForInit := SUPER^.SaveOnlineParametersForInit();
END_METHOD

PROPERTY SimulinkTime_Online : LREAL
GET
hResult := GetObjPara(16#00000005,sizeof(SimulinkTime_Online),adr(SimulinkTime_Online));
END_GET
SET
hResult := SetObjPara(16#00000005,sizeof(SimulinkTime_Online),adr(SimulinkTime_Online));
END_SET
END_PROPERTY

PROPERTY StepSize_Online : TctStepSizeType
GET
hResult := GetObjPara(16#00000002,sizeof(StepSize_Online),adr(StepSize_Online));
END_GET
SET
hResult := SetObjPara(16#00000002,sizeof(StepSize_Online),adr(StepSize_Online));
END_SET
END_PROPERTY

PROPERTY StepSize_Startup : TctStepSizeType
GET
StepSize_Startup := stInitData.StepSize;
END_GET
SET
stInitData.StepSize := StepSize_Startup;
END_SET
END_PROPERTY

{attribute 'object_name' := 'VerifyParameters'}
METHOD PRIVATE VerifyParameters : HRESULT
VAR
	moduleCallByParam: TctModuleCallByType;
END_VAR

IF (bParametersVerified) THEN
  VerifyParameters := Tc2_System.E_HRESULTAdsErr.HRESULT_ADS_NOERROR;
ELSE
  VerifyParameters := GetObjPara(stInitData.CallByHdr.indexOffset,SIZEOF(moduleCallByParam),ADR(moduleCallByParam));
  
  // check the "CallBy" parameter to be set to "Module"
  IF (SUCCEEDED(VerifyParameters) AND (moduleCallByParam <> TctModuleCallByType.Module)) THEN
      VerifyParameters := Tc2_System.E_HRESULTAdsErr.INVALIDPARM;
  END_IF
  
  // set the parameters verified flag
  bParametersVerified := SUCCEEDED(VerifyParameters);
END_IF
END_METHOD

END_FUNCTION_BLOCK

// ---- DUTs/Filter_Current/FB_Filter_Current_Hexapod_Robot.TcPOU
{attribute 'TcDependOnClassFactory' := 'Filter_Current_Hexapod_Robot'}
FUNCTION_BLOCK FB_Filter_Current_Hexapod_Robot EXTENDS FB_TcMatSimObject
VAR_INPUT
	stInput: ST_Filter_Current_Hexapod_Robot_Input;
END_VAR
VAR_OUTPUT
	stOutput: ST_Filter_Current_Hexapod_Robot_Output;
END_VAR
VAR
	stInitData: ST_Filter_Current_Hexapod_Robot_InitData;
	arrDataAreas: ARRAY[1..2] OF ST_TcMatSimObjectDataAreaInfo;
	bParametersVerified: BOOL;
END_VAR

PROPERTY CallBy_Online : TctModuleCallByType
GET
hResult := GetObjPara(16#00000000,sizeof(CallBy_Online),adr(CallBy_Online));
END_GET
SET
hResult := SetObjPara(16#00000000,sizeof(CallBy_Online),adr(CallBy_Online));
END_SET
END_PROPERTY

PROPERTY CallBy_Startup : TctModuleCallByType
GET
CallBy_Startup := stInitData.CallBy;
END_GET
SET
stInitData.CallBy := CallBy_Startup;
END_SET
END_PROPERTY

PROPERTY ContextInfoArr_0_TaskCycleTimeNs_Online : UDINT
GET
hResult := GetObjPara(16#03002080,sizeof(ContextInfoArr_0_TaskCycleTimeNs_Online),adr(ContextInfoArr_0_TaskCycleTimeNs_Online));
END_GET
SET
hResult := SetObjPara(16#03002080,sizeof(ContextInfoArr_0_TaskCycleTimeNs_Online),adr(ContextInfoArr_0_TaskCycleTimeNs_Online));
END_SET
END_PROPERTY

PROPERTY ContextInfoArr_0_TaskCycleTimeNs_Startup : UDINT
GET
ContextInfoArr_0_TaskCycleTimeNs_Startup := stInitData.ContextInfoArr_0_TaskCycleTimeNs;
END_GET
SET
stInitData.ContextInfoArr_0_TaskCycleTimeNs := ContextInfoArr_0_TaskCycleTimeNs_Startup;
END_SET
END_PROPERTY

PROPERTY ContextInfoArr_0_TaskOid_Online : OTCID
GET
hResult := GetObjPara(16#03002060,sizeof(ContextInfoArr_0_TaskOid_Online),adr(ContextInfoArr_0_TaskOid_Online));
END_GET
SET
hResult := SetObjPara(16#03002060,sizeof(ContextInfoArr_0_TaskOid_Online),adr(ContextInfoArr_0_TaskOid_Online));
END_SET
END_PROPERTY

PROPERTY ContextInfoArr_0_TaskOid_Startup : OTCID
GET
ContextInfoArr_0_TaskOid_Startup := stInitData.ContextInfoArr_0_TaskOid;
END_GET
SET
stInitData.ContextInfoArr_0_TaskOid := ContextInfoArr_0_TaskOid_Startup;
END_SET
END_PROPERTY

PROPERTY ContextInfoArr_0_TaskPort_Online : UINT
GET
hResult := GetObjPara(16#03002090,sizeof(ContextInfoArr_0_TaskPort_Online),adr(ContextInfoArr_0_TaskPort_Online));
END_GET
SET
hResult := SetObjPara(16#03002090,sizeof(ContextInfoArr_0_TaskPort_Online),adr(ContextInfoArr_0_TaskPort_Online));
END_SET
END_PROPERTY

PROPERTY ContextInfoArr_0_TaskPort_Startup : UINT
GET
ContextInfoArr_0_TaskPort_Startup := stInitData.ContextInfoArr_0_TaskPort;
END_GET
SET
stInitData.ContextInfoArr_0_TaskPort := ContextInfoArr_0_TaskPort_Startup;
END_SET
END_PROPERTY

PROPERTY ContextInfoArr_0_TaskPriority_Online : UDINT
GET
hResult := GetObjPara(16#03002070,sizeof(ContextInfoArr_0_TaskPriority_Online),adr(ContextInfoArr_0_TaskPriority_Online));
END_GET
SET
hResult := SetObjPara(16#03002070,sizeof(ContextInfoArr_0_TaskPriority_Online),adr(ContextInfoArr_0_TaskPriority_Online));
END_SET
END_PROPERTY

PROPERTY ContextInfoArr_0_TaskPriority_Startup : UDINT
GET
ContextInfoArr_0_TaskPriority_Startup := stInitData.ContextInfoArr_0_TaskPriority;
END_GET
SET
stInitData.ContextInfoArr_0_TaskPriority := ContextInfoArr_0_TaskPriority_Startup;
END_SET
END_PROPERTY

PROPERTY ContextInfoArr_0_TaskSortOrder_Online : UDINT
GET
hResult := GetObjPara(16#030020b0,sizeof(ContextInfoArr_0_TaskSortOrder_Online),adr(ContextInfoArr_0_TaskSortOrder_Online));
END_GET
SET
hResult := SetObjPara(16#030020b0,sizeof(ContextInfoArr_0_TaskSortOrder_Online),adr(ContextInfoArr_0_TaskSortOrder_Online));
END_SET
END_PROPERTY

PROPERTY ContextInfoArr_0_TaskSortOrder_Startup : UDINT
GET
ContextInfoArr_0_TaskSortOrder_Startup := stInitData.ContextInfoArr_0_TaskSortOrder;
END_GET
SET
stInitData.ContextInfoArr_0_TaskSortOrder := ContextInfoArr_0_TaskSortOrder_Startup;
END_SET
END_PROPERTY

PROPERTY CycleUpdateExecuted_Online : BOOL
GET
hResult := GetObjPara(16#00000004,sizeof(CycleUpdateExecuted_Online),adr(CycleUpdateExecuted_Online));
END_GET
SET
hResult := SetObjPara(16#00000004,sizeof(CycleUpdateExecuted_Online),adr(CycleUpdateExecuted_Online));
END_SET
END_PROPERTY

METHOD Execute : HRESULT

IF (SUCCEEDED(hResult)) THEN
  hResult := VerifyParameters();
END_IF

	// update DataArea information
SetDataAreaInfo(ADR(arrDataAreas),2);
	
	// call base method
Execute := SUPER^.Execute();
END_METHOD

PROPERTY ExecuteModelCode_Online : BOOL
GET
hResult := GetObjPara(16#00000008,sizeof(ExecuteModelCode_Online),adr(ExecuteModelCode_Online));
END_GET
SET
hResult := SetObjPara(16#00000008,sizeof(ExecuteModelCode_Online),adr(ExecuteModelCode_Online));
END_SET
END_PROPERTY

PROPERTY ExecuteModelCode_Startup : BOOL
GET
ExecuteModelCode_Startup := stInitData.ExecuteModelCode;
END_GET
SET
stInitData.ExecuteModelCode := ExecuteModelCode_Startup;
END_SET
END_PROPERTY

PROPERTY ExecutionSequence_Online : TctModuleExecutionSequenceType
GET
hResult := GetObjPara(16#00000001,sizeof(ExecutionSequence_Online),adr(ExecutionSequence_Online));
END_GET
SET
hResult := SetObjPara(16#00000001,sizeof(ExecutionSequence_Online),adr(ExecutionSequence_Online));
END_SET
END_PROPERTY

PROPERTY ExecutionSequence_Startup : TctModuleExecutionSequenceType
GET
ExecutionSequence_Startup := stInitData.ExecutionSequence;
END_GET
SET
stInitData.ExecutionSequence := ExecutionSequence_Startup;
END_SET
END_PROPERTY

METHOD FB_init : BOOL
VAR_INPUT
	/// if TRUE, the retain variables are initialized (warm start / cold start)
	bInitRetains: BOOL;
	/// if TRUE, the instance afterwards gets moved into the copy code (online change)
	bInCopyCode: BOOL;
	oid: OTCID;
END_VAR
VAR
	clsId: CLSID;
END_VAR

// initialize flags
bParametersVerified := false;
                    
// set module class id for compatibility check
clsId.Data1 := 16#4ef20903;
clsId.Data2 := 16#d648;
clsId.Data3 := 16#49c7;
clsId.Data4[0] := 16#a9;
clsId.Data4[1] := 16#06;
clsId.Data4[2] := 16#8c;
clsId.Data4[3] := 16#fc;
clsId.Data4[4] := 16#20;
clsId.Data4[5] := 16#50;
clsId.Data4[6] := 16#7f;
clsId.Data4[7] := 16#b3;

AssignClassId(clsId);
                    
// initialize InitData structure with default values              
stInitData.CallByHdr.indexGroup := 0;
stInitData.CallByHdr.indexOffset := 16#00000000;
stInitData.CallByHdr.cbData := SIZEOF(stInitData.CallBy);
stInitData.CallBy := TctModuleCallByType.Module;
stInitData.ExecutionSequenceHdr.indexGroup := 0;
stInitData.ExecutionSequenceHdr.indexOffset := 16#00000001;
stInitData.ExecutionSequenceHdr.cbData := SIZEOF(stInitData.ExecutionSequence);
stInitData.ExecutionSequence := TctModuleExecutionSequenceType.StateUpdateAfterOutputMapping;
stInitData.StepSizeHdr.indexGroup := 0;
stInitData.StepSizeHdr.indexOffset := 16#00000002;
stInitData.StepSizeHdr.cbData := SIZEOF(stInitData.StepSize);
stInitData.StepSize := TctStepSizeType.UseTaskCycleTime;
stInitData.ExecuteModelCodeHdr.indexGroup := 0;
stInitData.ExecuteModelCodeHdr.indexOffset := 16#00000008;
stInitData.ExecuteModelCodeHdr.cbData := SIZEOF(stInitData.ExecuteModelCode);
stInitData.ExecuteModelCode := 1;
stInitData.ModelParametersHdr.indexGroup := 0;
stInitData.ModelParametersHdr.indexOffset := 16#83000000;
stInitData.ModelParametersHdr.cbData := SIZEOF(stInitData.ModelParameters);
stInitData.ModelParameters.DiscreteFilter_NumCoef[0] := 1.25663706143591720e+01;
stInitData.ModelParameters.DiscreteFilter_NumCoef[1] := 1.25663706143591720e+01;
stInitData.ModelParameters.DiscreteFilter_DenCoef[0] := 2.01256637061435910e+03;
stInitData.ModelParameters.DiscreteFilter_DenCoef[1] := -1.98743362938564090e+03;
stInitData.ModelParameters.DiscreteFilter_InitialStates := 0.00000000000000000e+00;
stInitData.ModelParameters.DiscreteFilter1_NumCoef[0] := 1.25663706143591720e+01;
stInitData.ModelParameters.DiscreteFilter1_NumCoef[1] := 1.25663706143591720e+01;
stInitData.ModelParameters.DiscreteFilter1_DenCoef[0] := 2.01256637061435910e+03;
stInitData.ModelParameters.DiscreteFilter1_DenCoef[1] := -1.98743362938564090e+03;
stInitData.ModelParameters.DiscreteFilter1_InitialStates := 0.00000000000000000e+00;
stInitData.ModelParameters.DiscreteFilter2_NumCoef[0] := 1.25663706143591720e+01;
stInitData.ModelParameters.DiscreteFilter2_NumCoef[1] := 1.25663706143591720e+01;
stInitData.ModelParameters.DiscreteFilter2_DenCoef[0] := 2.01256637061435910e+03;
stInitData.ModelParameters.DiscreteFilter2_DenCoef[1] := -1.98743362938564090e+03;
stInitData.ModelParameters.DiscreteFilter2_InitialStates := 0.00000000000000000e+00;
stInitData.ModelParameters.DiscreteFilter3_NumCoef[0] := 1.25663706143591720e+01;
stInitData.ModelParameters.DiscreteFilter3_NumCoef[1] := 1.25663706143591720e+01;
stInitData.ModelParameters.DiscreteFilter3_DenCoef[0] := 2.01256637061435910e+03;
stInitData.ModelParameters.DiscreteFilter3_DenCoef[1] := -1.98743362938564090e+03;
stInitData.ModelParameters.DiscreteFilter3_InitialStates := 0.00000000000000000e+00;
stInitData.ModelParameters.DiscreteFilter4_NumCoef[0] := 1.25663706143591720e+01;
stInitData.ModelParameters.DiscreteFilter4_NumCoef[1] := 1.25663706143591720e+01;
stInitData.ModelParameters.DiscreteFilter4_DenCoef[0] := 2.01256637061435910e+03;
stInitData.ModelParameters.DiscreteFilter4_DenCoef[1] := -1.98743362938564090e+03;
stInitData.ModelParameters.DiscreteFilter4_InitialStates := 0.00000000000000000e+00;
stInitData.ModelParameters.DiscreteFilter5_NumCoef[0] := 1.25663706143591720e+01;
stInitData.ModelParameters.DiscreteFilter5_NumCoef[1] := 1.25663706143591720e+01;
stInitData.ModelParameters.DiscreteFilter5_DenCoef[0] := 2.01256637061435910e+03;
stInitData.ModelParameters.DiscreteFilter5_DenCoef[1] := -1.98743362938564090e+03;
stInitData.ModelParameters.DiscreteFilter5_InitialStates := 0.00000000000000000e+00;
stInitData.ModelParameters.DiscreteFilter6_NumCoef[0] := 1.25663706143591720e+01;
stInitData.ModelParameters.DiscreteFilter6_NumCoef[1] := 1.25663706143591720e+01;
stInitData.ModelParameters.DiscreteFilter6_DenCoef[0] := 2.01256637061435910e+03;
stInitData.ModelParameters.DiscreteFilter6_DenCoef[1] := -1.98743362938564090e+03;
stInitData.ModelParameters.DiscreteFilter6_InitialStates := 0.00000000000000000e+00;
stInitData.ModelParameters.DiscreteFilter7_NumCoef[0] := 1.25663706143591720e+01;
stInitData.ModelParameters.DiscreteFilter7_NumCoef[1] := 1.25663706143591720e+01;
stInitData.ModelParameters.DiscreteFilter7_DenCoef[0] := 2.01256637061435910e+03;
stInitData.ModelParameters.DiscreteFilter7_DenCoef[1] := -1.98743362938564090e+03;
stInitData.ModelParameters.DiscreteFilter7_InitialStates := 0.00000000000000000e+00;
stInitData.ModelParameters.DiscreteFilter8_NumCoef[0] := 1.25663706143591720e+01;
stInitData.ModelParameters.DiscreteFilter8_NumCoef[1] := 1.25663706143591720e+01;
stInitData.ModelParameters.DiscreteFilter8_DenCoef[0] := 2.01256637061435910e+03;
stInitData.ModelParameters.DiscreteFilter8_DenCoef[1] := -1.98743362938564090e+03;
stInitData.ModelParameters.DiscreteFilter8_InitialStates := 0.00000000000000000e+00;
stInitData.ModelParameters.DiscreteFilter9_NumCoef[0] := 1.25663706143591720e+01;
stInitData.ModelParameters.DiscreteFilter9_NumCoef[1] := 1.25663706143591720e+01;
stInitData.ModelParameters.DiscreteFilter9_DenCoef[0] := 2.01256637061435910e+03;
stInitData.ModelParameters.DiscreteFilter9_DenCoef[1] := -1.98743362938564090e+03;
stInitData.ModelParameters.DiscreteFilter9_InitialStates := 0.00000000000000000e+00;
stInitData.ModelParameters.DiscreteFilter10_NumCoef[0] := 1.25663706143591720e+01;
stInitData.ModelParameters.DiscreteFilter10_NumCoef[1] := 1.25663706143591720e+01;
stInitData.ModelParameters.DiscreteFilter10_DenCoef[0] := 2.01256637061435910e+03;
stInitData.ModelParameters.DiscreteFilter10_DenCoef[1] := -1.98743362938564090e+03;
stInitData.ModelParameters.DiscreteFilter10_InitialStates := 0.00000000000000000e+00;
stInitData.ModelParameters.DiscreteFilter11_NumCoef[0] := 1.25663706143591720e+01;
stInitData.ModelParameters.DiscreteFilter11_NumCoef[1] := 1.25663706143591720e+01;
stInitData.ModelParameters.DiscreteFilter11_DenCoef[0] := 2.01256637061435910e+03;
stInitData.ModelParameters.DiscreteFilter11_DenCoef[1] := -1.98743362938564090e+03;
stInitData.ModelParameters.DiscreteFilter11_InitialStates := 0.00000000000000000e+00;
stInitData.ModelParameters.DiscreteFilter12_NumCoef[0] := 1.25663706143591720e+01;
stInitData.ModelParameters.DiscreteFilter12_NumCoef[1] := 1.25663706143591720e+01;
stInitData.ModelParameters.DiscreteFilter12_DenCoef[0] := 2.01256637061435910e+03;
stInitData.ModelParameters.DiscreteFilter12_DenCoef[1] := -1.98743362938564090e+03;
stInitData.ModelParameters.DiscreteFilter12_InitialStates := 0.00000000000000000e+00;
stInitData.ModelParameters.DiscreteFilter13_NumCoef[0] := 1.25663706143591720e+01;
stInitData.ModelParameters.DiscreteFilter13_NumCoef[1] := 1.25663706143591720e+01;
stInitData.ModelParameters.DiscreteFilter13_DenCoef[0] := 2.01256637061435910e+03;
stInitData.ModelParameters.DiscreteFilter13_DenCoef[1] := -1.98743362938564090e+03;
stInitData.ModelParameters.DiscreteFilter13_InitialStates := 0.00000000000000000e+00;
stInitData.ModelParameters.DiscreteFilter14_NumCoef[0] := 1.25663706143591720e+01;
stInitData.ModelParameters.DiscreteFilter14_NumCoef[1] := 1.25663706143591720e+01;
stInitData.ModelParameters.DiscreteFilter14_DenCoef[0] := 2.01256637061435910e+03;
stInitData.ModelParameters.DiscreteFilter14_DenCoef[1] := -1.98743362938564090e+03;
stInitData.ModelParameters.DiscreteFilter14_InitialStates := 0.00000000000000000e+00;
stInitData.ModelParameters.DiscreteFilter15_NumCoef[0] := 1.25663706143591720e+01;
stInitData.ModelParameters.DiscreteFilter15_NumCoef[1] := 1.25663706143591720e+01;
stInitData.ModelParameters.DiscreteFilter15_DenCoef[0] := 2.01256637061435910e+03;
stInitData.ModelParameters.DiscreteFilter15_DenCoef[1] := -1.98743362938564090e+03;
stInitData.ModelParameters.DiscreteFilter15_InitialStates := 0.00000000000000000e+00;
stInitData.ModelParameters.DiscreteFilter16_NumCoef[0] := 1.25663706143591720e+01;
stInitData.ModelParameters.DiscreteFilter16_NumCoef[1] := 1.25663706143591720e+01;
stInitData.ModelParameters.DiscreteFilter16_DenCoef[0] := 2.01256637061435910e+03;
stInitData.ModelParameters.DiscreteFilter16_DenCoef[1] := -1.98743362938564090e+03;
stInitData.ModelParameters.DiscreteFilter16_InitialStates := 0.00000000000000000e+00;
stInitData.ModelParameters.DiscreteFilter17_NumCoef[0] := 1.25663706143591720e+01;
stInitData.ModelParameters.DiscreteFilter17_NumCoef[1] := 1.25663706143591720e+01;
stInitData.ModelParameters.DiscreteFilter17_DenCoef[0] := 2.01256637061435910e+03;
stInitData.ModelParameters.DiscreteFilter17_DenCoef[1] := -1.98743362938564090e+03;
stInitData.ModelParameters.DiscreteFilter17_InitialStates := 0.00000000000000000e+00;
stInitData.ContextInfoArr_0_TaskOidHdr.indexGroup := 0;
stInitData.ContextInfoArr_0_TaskOidHdr.indexOffset := 16#03002060;
stInitData.ContextInfoArr_0_TaskOidHdr.cbData := SIZEOF(stInitData.ContextInfoArr_0_TaskOid);
stInitData.ContextInfoArr_0_TaskPriorityHdr.indexGroup := 0;
stInitData.ContextInfoArr_0_TaskPriorityHdr.indexOffset := 16#03002070;
stInitData.ContextInfoArr_0_TaskPriorityHdr.cbData := SIZEOF(stInitData.ContextInfoArr_0_TaskPriority);
stInitData.ContextInfoArr_0_TaskCycleTimeNsHdr.indexGroup := 0;
stInitData.ContextInfoArr_0_TaskCycleTimeNsHdr.indexOffset := 16#03002080;
stInitData.ContextInfoArr_0_TaskCycleTimeNsHdr.cbData := SIZEOF(stInitData.ContextInfoArr_0_TaskCycleTimeNs);
stInitData.ContextInfoArr_0_TaskPortHdr.indexGroup := 0;
stInitData.ContextInfoArr_0_TaskPortHdr.indexOffset := 16#03002090;
stInitData.ContextInfoArr_0_TaskPortHdr.cbData := SIZEOF(stInitData.ContextInfoArr_0_TaskPort);
stInitData.ContextInfoArr_0_TaskSortOrderHdr.indexGroup := 0;
stInitData.ContextInfoArr_0_TaskSortOrderHdr.indexOffset := 16#030020b0;
stInitData.ContextInfoArr_0_TaskSortOrderHdr.cbData := SIZEOF(stInitData.ContextInfoArr_0_TaskSortOrder);
stInitData.Header.cbData := SIZEOF(stInitData)-SIZEOF(stInitData.Header);
stInitData.Header.uiElmCnt := 10;


// set pointer to InitData structure
SetInitDataInfo(ADR(stInitData));

// set DataArea information
SetDataAreaInfo(ADR(arrDataAreas),2);
arrDataAreas[1].nDataAreaId := 0;
arrDataAreas[1].nSize := SIZEOF(stInput);
arrDataAreas[1].pPlcVar := ADR(stInput);
arrDataAreas[1].pModuleProcImg := 0;
arrDataAreas[1].eDataAreaType := E_TcMatSimDataAreaType.InputDst;
arrDataAreas[2].nDataAreaId := 1;
arrDataAreas[2].nSize := SIZEOF(stOutput);
arrDataAreas[2].pPlcVar := ADR(stOutput);
arrDataAreas[2].pModuleProcImg := 0;
arrDataAreas[2].eDataAreaType := E_TcMatSimDataAreaType.OutputSrc;


// initialize basic interface pointers and return
FB_init := SUCCEEDED(Init(oid));
END_METHOD

PROPERTY InitData : ST_Filter_Current_Hexapod_Robot_InitData
GET
InitData := stInitData;
END_GET
SET
stInitData := InitData;
END_SET
END_PROPERTY

PROPERTY Input_Online : ExtU_Filter_Current_Hexapod_R_T
GET
hResult := GetObjPara(16#80000000,sizeof(Input_Online),adr(Input_Online));
END_GET
SET
hResult := SetObjPara(16#80000000,sizeof(Input_Online),adr(Input_Online));
END_SET
END_PROPERTY

{attribute 'object_name' := 'Internal_SetObjState'}
METHOD PROTECTED Internal_SetObjState
VAR_INPUT
	hr: REFERENCE TO HRESULT;
	nextState: TCOM_STATE;
END_VAR

// update pointer to InitData structure
SetInitDataInfo(ADR(stInitData));
// call base method
SUPER^.Internal_SetObjState(hr,nextState);
END_METHOD

PROPERTY MdlInitialized_Online : BOOL
GET
hResult := GetObjPara(16#00000003,sizeof(MdlInitialized_Online),adr(MdlInitialized_Online));
END_GET
SET
hResult := SetObjPara(16#00000003,sizeof(MdlInitialized_Online),adr(MdlInitialized_Online));
END_SET
END_PROPERTY

PROPERTY ModelParameters_Online : P_Filter_Current_Hexapod_Robo_T
GET
hResult := GetObjPara(16#83000000,sizeof(ModelParameters_Online),adr(ModelParameters_Online));
END_GET
SET
hResult := SetObjPara(16#83000000,sizeof(ModelParameters_Online),adr(ModelParameters_Online));
END_SET
END_PROPERTY

PROPERTY ModelParameters_Startup : P_Filter_Current_Hexapod_Robo_T
GET
ModelParameters_Startup := stInitData.ModelParameters;
END_GET
SET
stInitData.ModelParameters := ModelParameters_Startup;
END_SET
END_PROPERTY

PROPERTY ModuleBuildInfo_Online : TctModuleBuildInfoType
GET
hResult := GetObjPara(16#00000007,sizeof(ModuleBuildInfo_Online),adr(ModuleBuildInfo_Online));
END_GET
SET
hResult := SetObjPara(16#00000007,sizeof(ModuleBuildInfo_Online),adr(ModuleBuildInfo_Online));
END_SET
END_PROPERTY

PROPERTY ModuleInfo_Online : TctModuleInfoType
GET
hResult := GetObjPara(16#00000006,sizeof(ModuleInfo_Online),adr(ModuleInfo_Online));
END_GET
SET
hResult := SetObjPara(16#00000006,sizeof(ModuleInfo_Online),adr(ModuleInfo_Online));
END_SET
END_PROPERTY

{attribute 'object_name' := 'SaveOnlineParametersForInit'}
METHOD SaveOnlineParametersForInit : HRESULT
VAR
	idx: UINT;
	pInitElemHdr: POINTER TO TComInitDataElmHdr;
	pData: PVOID;
	nData: UDINT;
END_VAR
VAR CONSTANT
	nInitDataAlignment: UDINT := 4;
END_VAR

// update pointer to InitData structure
SetInitDataInfo(ADR(stInitData));
// call base method
SaveOnlineParametersForInit := SUPER^.SaveOnlineParametersForInit();
END_METHOD

PROPERTY SimulinkTime_Online : LREAL
GET
hResult := GetObjPara(16#00000005,sizeof(SimulinkTime_Online),adr(SimulinkTime_Online));
END_GET
SET
hResult := SetObjPara(16#00000005,sizeof(SimulinkTime_Online),adr(SimulinkTime_Online));
END_SET
END_PROPERTY

PROPERTY StepSize_Online : TctStepSizeType
GET
hResult := GetObjPara(16#00000002,sizeof(StepSize_Online),adr(StepSize_Online));
END_GET
SET
hResult := SetObjPara(16#00000002,sizeof(StepSize_Online),adr(StepSize_Online));
END_SET
END_PROPERTY

PROPERTY StepSize_Startup : TctStepSizeType
GET
StepSize_Startup := stInitData.StepSize;
END_GET
SET
stInitData.StepSize := StepSize_Startup;
END_SET
END_PROPERTY

{attribute 'object_name' := 'VerifyParameters'}
METHOD PRIVATE VerifyParameters : HRESULT
VAR
	moduleCallByParam: TctModuleCallByType;
END_VAR

IF (bParametersVerified) THEN
  VerifyParameters := Tc2_System.E_HRESULTAdsErr.HRESULT_ADS_NOERROR;
ELSE
  VerifyParameters := GetObjPara(stInitData.CallByHdr.indexOffset,SIZEOF(moduleCallByParam),ADR(moduleCallByParam));
  
  // check the "CallBy" parameter to be set to "Module"
  IF (SUCCEEDED(VerifyParameters) AND (moduleCallByParam <> TctModuleCallByType.Module)) THEN
      VerifyParameters := Tc2_System.E_HRESULTAdsErr.INVALIDPARM;
  END_IF
  
  // set the parameters verified flag
  bParametersVerified := SUCCEEDED(VerifyParameters);
END_IF
END_METHOD

END_FUNCTION_BLOCK

// ---- POUs/MAIN.TcPOU
PROGRAM MAIN
VAR_INPUT
	// ===================模块动作信号(按动作先后排列)==========
	Power_Execute 		: BOOL;							// 上电使能控制信号
	Axis_Power			: ARRAY[1..18] OF BOOL;			// 单电机使能
	Robot_Power			: BOOL;							// 机器人所有电机使能
	
	Home_Execute		: BOOL;							// 设置零点程序使能
	//Axis_Start_Back 	: ARRAY[1..18] OF BOOL;			// 单电机找零回退信号
	//Robot_Start_Back	: BOOL;							// 机器人所有电机回退信号
	Leg_Home_Set		: ARRAY[1..6] OF BOOL;	
	Axis_Home_Set		: ARRAY[1..18] OF BOOL;			// 单电机设定零点信号
	Robot_Home_Set		: BOOL;							// 机器人所有电机设定零点信号
	//Home_Set_Position	: ARRAY[1..18] OF LREAL;		// 找到零点后电机到达的位置
	//Delay_On			: ARRAY[1..18] OF BOOL;
	//TON1				: TON;
	
	Move_Execute		: BOOL;							// 绝对运动使能信号
	Robot_Stand_Execute	: BOOL;							// 机器人站立程序使能	
	Axis_Absolute_Eable	: ARRAY[1..18] OF BOOL;			// 单电机绝对运动使能信号
	Robot_Absolute_Eable: ARRAY[1..18] OF BOOL;			// 机器人站立使能信号
	Axis_Move_Position	: ARRAY[1..18] OF LREAL;		// 电机绝对运动位置			
	
	Reset_Execute		: BOOL;							// 电机驱动重置动作发生使能
	Axis_Reset			: ARRAY[1..18] OF BOOL;			// 单电机驱动重置信号使能
	Robot_Reset			: BOOL;							// 机器人整体电机驱动重置
	//Axis_ResetDone		: ARRAY[1..18] OF BOOL;			// 单电机驱动重置完成

END_VAR
VAR
// =======================NC轴变量==========================
	//Leg_Robot			: ARRAY[1..6] OF Hexapod_Leg;	// 定义六足的腿
	Axis_Robot			: ARRAY[1..18] OF Axis;			// 定义六足轴参量(可以调整数据上限来调整电机数目)
	Axis_Delay			: Delay;						// 延迟程序
	Leg_Number			: INT;							// 定义机器人腿数
	Axis_Number 		: INT;							// 定义轴数目
	
	// ===================状态监测变量=======================
	Power_Status	: ARRAY[1..18] OF BOOL;				// 上电监测信号
	Leg_Home_Done	: ARRAY[1..6] OF BOOL;
	Home_Done		: ARRAY[1..18] OF BOOL;				// 找零监测信号
	MoveAbsoluteDone: ARRAY[1..18] OF BOOL;				// 电机运动监测信号
	
	Robot_Error		: BOOL;								// 机器人电机错误信号
	Axis_Error		: ARRAY[1..18] OF BOOL;				// 电机错误监测信号
	Axis_ErrorID	: ARRAY[1..18] OF UDINT;			// 电机错误号码监测信号
	
	Axis_ActPostion	: ARRAY[1..18] OF LREAL;			// 电机轴实际位置
	
	// =======================模块中间变量======================
	//HomeDone_Number	: LREAL :=0;					//完成找零的轴数
	//ExSetPoint_Position	: ARRAY[1..18] OF LREAL;		// 外部信号位置
	//t					: LREAL :=0;
	
	// =======================驱动器信号监测====================
	Current_Turque_Value  AT%IW0 : ARRAY[1..18] OF INT ;//电流、力矩相关值
	Current_Before_Mapping	: ARRAY[1..18] OF LREAL ;	// 将Current_Turque_Value转换数制
	Max_Turque_Value 		: INT ;						// 设置最大力矩边界值
	Mapping_Current			: Variable_Control_Mapping_Model;	// 变量映射	
	Current_After_Mapping	: ARRAY[1..18] OF LREAL;	// 映射后的原始电流值
	
	// ====================Simulink模块相关=====================  
  //Filter_Current  : FB_Filter_Current_Hexapod_Robot(oid:=16#01010030);
  //Current_Turque_Filter  : ARRAY[1..18] OF LREAL;
END_VAR

// =======================子程序使能(永久运行)===================
Variable_Monitor();			// 变量监测子程序使能
Logic_Control();			// 逻辑控制子程序使能
Variable_Set();				// 各动作速度子程序使能
Leg_Action();				// 单腿运动子程序使能
Robot_Action();				// 机器人整体运动子程序使能

// =====================电机驱动重置=============================
IF Reset_Execute THEN
	FOR Axis_Number := 1 TO 18 {BY 1} DO
		Axis_Robot[Axis_Number].Reset(Drive_Reset:= Axis_Reset[Axis_Number]);
	END_FOR
END_IF

// =======================电机上电===============================
IF Power_Execute THEN
	FOR Axis_Number := 1 TO 18 {BY 1} DO
		Axis_Robot[Axis_Number].Power(Axis_Enable:= Axis_Power[Axis_Number]);
	END_FOR
END_IF

// =======================找零程序===============================
IF Home_Execute THEN
	FOR Axis_Number := 1 TO 18 {BY 1} DO
		Axis_Robot[Axis_Number].Home(Drive_Home:= Axis_Home_Set[Axis_Number]);
	END_FOR
END_IF

// =======================站立程序===============================
IF Move_Execute THEN
	FOR Axis_Number := 1 TO 18 {BY 1} DO
		Axis_Robot[Axis_Number].Move_Absolute(	Drive_Move_Absolute:= Axis_Absolute_Eable[Axis_Number], 
												Absolute_Position:= Axis_Move_Position[Axis_Number]);
	END_FOR
END_IF

ACTION Leg_Action:
// ===================机器人单条腿找零程序====================
IF Home_Execute THEN
	FOR Leg_Number := 1 TO 6 {BY 1} DO
		IF Leg_Home_Set[Leg_Number] THEN		// 在可视化中，Leg_Home_Set为点动
			Axis_Home_Set[1+(Leg_Number-1)*3] := Leg_Home_Set[Leg_Number];
			Axis_Home_Set[2+(Leg_Number-1)*3] := Leg_Home_Set[Leg_Number];
			Axis_Home_Set[3+(Leg_Number-1)*3] := Leg_Home_Set[Leg_Number];
		ELSIF Home_Done[1+(Leg_Number-1)*3] AND Home_Done[2+(Leg_Number-1)*3] AND Home_Done[3+(Leg_Number-1)*3] THEN
			Leg_Home_Set[Leg_Number] := FALSE; 
		END_IF
	END_FOR
END_IF
END_ACTION

ACTION Logic_Control:
// =======================控制逻辑区==========================
// 保证所有的动作拥有合理的先后顺序，优化控制逻辑
// 也防止出现两个或两个以上动作同时进行的情况，保证控制安全

// ===================电机驱动重置逻辑========================
//FOR Axis_Number := 1 TO 18 {BY 1} DO
IF Axis_Error[1] OR Axis_Error[2] OR Axis_Error[3] OR Axis_Error[4] OR Axis_Error[5] OR Axis_Error[6]
	 OR Axis_Error[7] OR Axis_Error[8] OR Axis_Error[9] OR Axis_Error[10] OR Axis_Error[11] OR Axis_Error[12]
		OR Axis_Error[13] OR Axis_Error[14] OR Axis_Error[15] OR Axis_Error[16] OR Axis_Error[17] OR Axis_Error[18]
THEN
	Robot_Error := TRUE;
ELSE
	Robot_Error := FALSE;
END_IF
//END_FOR

IF Robot_Error THEN
	Reset_Execute := TRUE;
ELSIF NOT Robot_Error THEN
	Reset_Execute := FALSE;
ELSIF NOT Reset_Execute THEN
	Axis_Reset[Axis_Number] := FALSE;
	Axis_Robot[Axis_Number].Reset(Drive_Reset:= Axis_Reset[Axis_Number]);
END_IF

// =====================上电程序逻辑==========================
IF NOT Power_Execute THEN
	FOR Axis_Number := 1 TO 18 {BY 1} DO
		Axis_Power[Axis_Number] := FALSE;
		Axis_Robot[Axis_Number].Power(Axis_Enable:= Axis_Power[Axis_Number]);
	END_FOR
END_IF

// =====================找零程序逻辑==========================
IF Home_Execute THEN
	FOR Axis_Number := 1 TO 18 {BY 1} DO
		IF Home_Done[Axis_Number] THEN			// 	丝杠到达零点位置后，单电机标零使能位关闭			
			Axis_Home_Set[Axis_Number] :=0;	
			Axis_Robot[Axis_Number].Home(Drive_Home:= Axis_Home_Set[Axis_Number]);
		END_IF
	END_FOR
	Move_Execute :=0;							// 设定零点时，不能进行其他运动
	//ExSetPoint_Execute :=0;
ELSIF NOT Home_Execute THEN
	FOR Axis_Number := 1 TO 18 {BY 1} DO
		//Axis_Start_Back[Axis_Number] :=0;
		Axis_Home_Set[Axis_Number] := 0;
	END_FOR
END_IF

// =====================机器人站立逻辑==========================
IF Move_Execute THEN
	//Absolute_Eable := TRUE;
	Home_Execute := FALSE;						// 站立运动使能时，机器人调零必须结束
	//ExSetPoint_Execute :=0;						// 站立运动时，不能进行其他运动
	FOR Axis_Number := 1 TO 18 {BY 1} DO
		IF MoveAbsoluteDone[Axis_Number] THEN	// 	丝杠到达设定位置后，单电机绝对运动使能位关闭
			Axis_Absolute_Eable[Axis_Number] := FALSE;
		END_IF
	END_FOR
ELSIF NOT Move_Execute THEN						// 站立运动不使能,轴不能运动
	FOR Axis_Number := 1 TO 18 {BY 1} DO
		Axis_Absolute_Eable[Axis_Number] := FALSE;
		Axis_Robot[Axis_Number].Move_Absolute(	Drive_Move_Absolute:= Axis_Absolute_Eable[Axis_Number], 
												Absolute_Position:= Axis_Move_Position[Axis_Number]);
	END_FOR
END_IF
END_ACTION

ACTION Robot_Action:
// =================机器人整体运动命令区======================
// 六足所有电机整体控制

// ====================机器人驱动重置=========================
IF Robot_Reset THEN
	IF Reset_Execute THEN
		Axis_Reset[Axis_Number] := TRUE;
		FOR Axis_Number := 1 TO 18 {BY 1} DO
			Axis_Robot[Axis_Number].Reset(Drive_Reset:= Axis_Reset[Axis_Number]);
		END_FOR
	END_IF
END_IF	

// ===================机器人所有电机上电======================
IF Robot_Power THEN	
	IF Power_Execute THEN
		FOR Axis_Number := 1 TO 18 {BY 1} DO
			Axis_Power[Axis_Number] := TRUE ;
		END_FOR
	END_IF
END_IF
	
// ===================机器人找零程序=======================
IF Robot_Home_Set THEN				// 标零程序
	//Robot_Start_Back := FALSE;
	IF Home_Execute THEN
		Leg_Home_Set[3] := Leg_Home_Set[5] := Leg_Home_Set[1];	// 在整机调零时，1\3\5三条腿同时调零；
		Leg_Home_Set[4] := Leg_Home_Set[6] := Leg_Home_Set[2];	// 在整机调零时，2\4\6三条腿同时调零；
	ELSIF NOT Home_Execute THEN
		FOR Leg_Number := 1 TO 6 {BY 1} DO
			Leg_Home_Set[Leg_Number] := FALSE;
		END_FOR
	END_IF
ELSIF NOT Robot_Home_Set AND NOT Home_Execute THEN
	FOR Axis_Number := 1 TO 18 {BY 1} DO
	Axis_Home_Set[Axis_Number] := FALSE;
	END_FOR
END_IF

// =====================站立程序===============================
IF Robot_Stand_Execute THEN
	IF Move_Execute THEN
		FOR Axis_Number := 1 TO 18 {BY 1} DO
			IF MoveAbsoluteDone[Axis_Number] THEN		// 	丝杠到达设定位置后，单电机绝对运动使能位关闭
				Axis_Absolute_Eable[Axis_Number] := FALSE;
			ELSE
				Axis_Absolute_Eable[Axis_Number] := TRUE;
			END_IF
		END_FOR
	END_IF
ELSIF NOT Robot_Stand_Execute AND NOT Move_Execute THEN 
	FOR Axis_Number := 1 TO 18 {BY 1} DO
		Axis_Absolute_Eable[Axis_Number] := FALSE;
	END_FOR
END_IF
END_ACTION

ACTION Variable_Monitor:
// =====================关键数据信号监测======================

// ==============最大力矩设置区(边界控制条件)=================
FOR Axis_Number := 1 TO 18 {BY 1} DO
	Axis_Robot[Axis_Number].Max_Turque_Value := Max_Turque_Value;
END_FOR

// =======================力矩检测区==========================
FOR Axis_Number := 1 TO 18 {BY 1} DO
	Axis_Robot[Axis_Number].Current_Turque_Value := Current_Turque_Value[Axis_Number];
	Current_Before_Mapping[Axis_Number] := INT_TO_LREAL(Current_Turque_Value[Axis_Number]);
END_FOR
Mapping_Current(Controller_Leg_Variable:= Current_Before_Mapping, Model_Leg_Variable=> Current_After_Mapping);

// ====================轴实际位置检测区=======================
FOR Axis_Number := 1 TO 18 {BY 1} DO
	Axis_ActPostion[Axis_Number] := Axis_Robot[Axis_Number].ActPosition;
END_FOR

// =======================上电状态检测区======================
FOR Axis_Number := 1 TO 18 {BY 1} DO
	Power_Status[Axis_Number] := Axis_Robot[Axis_Number].State_PowerStatus;
END_FOR

// =======================找零状态检测区======================
FOR Axis_Number := 1 TO 18 {BY 1} DO
	Home_Done[Axis_Number] := Axis_Robot[Axis_Number].State_HomeDone;
END_FOR

(*FOR Leg_Number := 1 TO 6 {BY 1} DO
	Leg_Home_Done[Leg_Number] := Leg_Robot[Axis_Number].State_HomeDone;
END_FOR*)

// ===================电机绝对运动状态检测区==================
FOR Axis_Number := 1 TO 18 {BY 1} DO
	MoveAbsoluteDone[Axis_Number] := Axis_Robot[Axis_Number].State_MoveAbsoluteDone;
END_FOR

// =======================电机错误检测区======================
FOR Axis_Number := 1 TO 18 {BY 1} DO
	Axis_Error[Axis_Number] := Axis_Robot[Axis_Number].Axis_Error;
	Axis_ErrorID[Axis_Number] := Axis_Robot[Axis_Number].Axis_ErrorID;
END_FOR
END_ACTION

ACTION Variable_Set:
// =======================速度规定区==========================
FOR Axis_Number := 1 TO 18 {BY 1} DO						//此时每一个电机的速度都是一样的
	Axis_Robot[Axis_Number].Home_Velocity 	:= 20;			//找零速度(Axis_Jog中的速度)
	Axis_Robot[Axis_Number].Move_Relative_Velocity	:=30;	//相对运动速度
END_FOR
IF Home_Execute THEN
	//IF Robot_Home_Set THEN
		Axis_Robot[1].Move_Absolute_Velocity :=17; Axis_Robot[3].Move_Absolute_Velocity :=17; Axis_Robot[4].Move_Absolute_Velocity :=16.74;
		Axis_Robot[6].Move_Absolute_Velocity :=16.74; Axis_Robot[7].Move_Absolute_Velocity :=17.3; Axis_Robot[9].Move_Absolute_Velocity :=17.3;
		Axis_Robot[10].Move_Absolute_Velocity :=16.95; Axis_Robot[12].Move_Absolute_Velocity :=16.95; Axis_Robot[13].Move_Absolute_Velocity :=17;
		Axis_Robot[15].Move_Absolute_Velocity :=17; Axis_Robot[16].Move_Absolute_Velocity :=17; Axis_Robot[18].Move_Absolute_Velocity :=17;
		Axis_Robot[2].Move_Absolute_Velocity :=20; Axis_Robot[5].Move_Absolute_Velocity :=19.8; Axis_Robot[8].Move_Absolute_Velocity :=20;
		Axis_Robot[11].Move_Absolute_Velocity :=20; Axis_Robot[14].Move_Absolute_Velocity :=20; Axis_Robot[17].Move_Absolute_Velocity :=20;
	//ELSIF NOT Robot_Home_Set THEN
		//FOR Axis_Number := 1 TO 18 {BY 1} DO
			//Axis_Robot[Axis_Number].Move_Absolute_Velocity	:=10;
		//END_FOR
	//END_IF
ELSE
	FOR Axis_Number := 1 TO 18 {BY 1} DO
			Axis_Robot[Axis_Number].Move_Absolute_Velocity	:=10;
	END_FOR
END_IF
	

// =======================位置规定区==========================
FOR Axis_Number := 1 TO 18 {BY 1} DO
	Axis_Move_Position[Axis_Number] := 160;
END_FOR

// =====================最大力矩规定区========================
Max_Turque_Value := 1000;

// ============电机设置零点后到达位置规定区(链接到Motor_Position_Generator)================
IF Home_Execute THEN
	FOR Axis_Number := 1 TO 18 {BY 1} DO
		Axis_Robot[Axis_Number].Home_Absolute_Position := Simulink_Model_Generator.Mapping_Position.Controller_Leg_Variable[Axis_Number];
	END_FOR
END_IF

// ===================程序与模型的变量链接===================
//FOR Axis_Number := 1 TO 18 {BY 1} DO
//	Simulink_Model_Generator.Filter_Current.stInput.Current_Motor[Axis_Number-1] := Current_Turque_Value[Axis_Number];
//END_FOR	
//Simulink_Model_Generator.Current_Turque_Filter := Simulink_Model_Generator.Filter_Current.stOutput.Current_Monitor;
END_ACTION

END_PROGRAM

// ---- DUTs/Axis/Axis.TcPOU
FUNCTION_BLOCK Axis
//VAR_INPUT	
//END_VAR
VAR_OUTPUT
	Axis_Error			: BOOL;				// Error signal
	Axis_ErrorID		: UDINT;			// Error ID
	Axis_Moves			: BOOL;				// Status of moving
END_VAR
VAR
	// =============== Done signals MC Block =================
	JogDone			    : BOOL;					// Status of function block MC_Jog
	ResetDone		    : BOOL;					// Status of function block MC_Reset
	HaltDone		    : BOOL;					// Status of function block MC_Halt
	HomeDone		    : BOOL;					// Status of function block MC_Home
  	MoveAbsoluteDone : BOOL;        // Status of function block MC_MoveAbsolute
  	ExtSetPiontDone 	: BOOL;         		// Status of function block MC_ExtSetPointGenDisable

	// =============== Control variables ======================
	//Home_Back_Start	: BOOL;
	//Drive_Home		: BOOL;
	
	// =============== State variables ========================
	Power_StatusEnable	: BOOL;					// Enable feedback
	
	// ============= Velocity, override ,Position==============
	Velocity_Jog		: LREAL;				// Jog velocity
	Velocity_Move		: LREAL;				// Target velocity
	Velocity_Home		: LREAL;				// Home velocity
	Velocity_Absolute	: LREAL;				// MoveAbsolute velocity
	Velocity_Relative	: LREAL;				// MoveRelative velocity
	fOverride 			: LREAL := 100.0;		// Override 100%
  Home_Position   : LREAL;        // The absolute position after Home will be
	
	// =============== Trigger function blocks ================
	
	TriggerHalt	: R_TRIG;				// Trigger to recognize rising edge of halt input
	TriggerReset : R_TRIG;				// Trigger to recognize rising edge of reset input
	
	// =============== Axis reference =========================
	AxisRef			: AXIS_REF;				// Axis reference (process data plc/nc)
	
	// =============== About axis turque ====================
	Axis_Current_Turque 	: INT;
  	Axis_Max_Turque       	: INT;

	// ================= Sensor FeedBack ====================
  	Proximity_Switch      : DINT;
	
	// =============== Motion function blocks =================
	Axis_Power 			: MC_Power;				// FB for enable and override			[上电]
	Axis_Home			: MC_Home;				// FB for axis home						[找零]
	Axis_Reset 			: MC_Reset;				// FB to reset axis						[复位]
	Axis_Jog			: MC_Jog;				// FB to jog axis						[点动]
	Axis_Stop 			: MC_Stop;				// FB to stop axis						[停止]
	Axis_Halt			: MC_Halt;				// FB to halt axis						[停止]
	Axis_Move			: MC_MoveVelocity;		// FB to move axis (velocity movement)	[匀速运动]
	Axis_MoveAbsolute 	: MC_MoveAbsolute;		// FB to move axis absolutely			[绝对位置运动]
	Axis_MoveRelative	: MC_MoveRelative;		// FB to move axis relatively			[相对位置运动]
  	Axis_ActPosition  : MC_ReadActualPosition; // FB to read the actual position of axis  [读取电机轴的实际位置]
	Axis_ActVelocity	: MC_ReadActualVelocity;// FB to read the actual Velocity of axis [读取电机轴的实际速度]
	Axis_Delay			: Delay;				// FB to operate the delay program		[延迟程序]
	Axis_ExtSetPiontEnable	: MC_ExtSetPointGenEnable;	// FB to enable extsetpoint		[外部函数发生使能]
	Axis_ExtSetPiontDisable	: MC_ExtSetPointGenDisable;	// FB to disable extsetpoint	[外部函数结束使能]
  
  // =============== Timer =================
  Delay         : TON;          //[定时器]
END_VAR

PROPERTY ActPosition : LREAL
GET
Axis_ActPosition( Axis:= AxisRef, Enable:= TRUE );
ActPosition := Axis_ActPosition.Position;
END_GET
END_PROPERTY

PROPERTY ActVelocity : LREAL
GET
Axis_ActVelocity( Axis:= AxisRef, Enable:= TRUE,  ActualVelocity=> ActVelocity);
END_GET
END_PROPERTY

PROPERTY Current_Turque_Value : INT
GET
Current_Turque_Value := Axis_Current_Turque;
END_GET
SET
Axis_Current_Turque := Current_Turque_Value;
END_SET
END_PROPERTY

METHOD ExtSetPoint
VAR_INPUT
	Drive_ExtSetPointEnable 	: BOOL;		// 使能外部信号开始信号
	Drive_ExtSetPointDisable 	: BOOL;		// 使能外部信号结束信号
	ExSetPosition				: LREAL;	// 外部信号位置
	//Axis_Current_Turque 		: INT;		// 边界条件：丝杠位置到达两端卡死
END_VAR
// =======================外部信号发生程序==========================

IF NOT Axis_ExtSetPiontEnable.Error THEN
	Axis_ExtSetPiontEnable(	Axis:= AxisRef, 
							Execute:= Drive_ExtSetPointEnable, 
							Position:= ExSetPosition, 
							PositionType:= POSITIONTYPE_ABSOLUTE );
END_IF

IF Axis_ExtSetPiontEnable.Done THEN
	ExtSetPiontDone := 1;
	MC_ExtSetPointGenFeed(	Position:= ExSetPosition, 
							Velocity:= 10, 
							Acceleration:= 10, 
							Direction:= 1, 		// 1 = positive direction
							Axis:= AxisRef );
END_IF	

IF NOT Axis_ExtSetPiontDisable.Error THEN 
	Axis_ExtSetPiontDisable(	Axis:= AxisRef, 
								Execute:= Drive_ExtSetPointDisable);
END_IF
								
IF Axis_ExtSetPiontEnable.Error OR Axis_ExtSetPiontDisable.Error OR ABS(Axis_Current_Turque) > Axis_Max_Turque THEN
	IF Axis_ExtSetPiontEnable.Error OR Axis_ExtSetPiontDisable.Error THEN
		Axis_Error		:= TRUE;
		Axis_ErrorID 	:= Axis_Home.ErrorID;
	END_IF
	Axis_ExtSetPiontEnable(	Axis:= AxisRef, 
							Execute:= 0 );
	Axis_ExtSetPiontDisable(	Axis:= AxisRef, 
								Execute:= 1);
END_IF
END_METHOD

METHOD Halt : BOOL
VAR_INPUT
	DriveHalt		: BOOL;					// Request stop
END_VAR
// =======================电机运动停止程序==========================

IF DriveHalt THEN
	// Move Execute FALSE
	Axis_Move(	Execute	:= FALSE,
				Axis 	:= AxisRef);
ELSE
	// Reset done signal
	HaltDone := FALSE;
END_IF

// Trigger
TriggerHalt(CLK := DriveHalt);

IF TriggerHalt.Q THEN
	Axis_Halt(	Execute	:= TRUE,
				Axis 	:= AxisRef);
ELSE
	Axis_Halt(Axis := AxisRef);
END_IF

// Done / Error / Command aborted
IF Axis_Halt.Done OR Axis_Halt.Error OR Axis_Halt.CommandAborted THEN
	Axis_Error		:= Axis_Halt.Error;
	Axis_ErrorID 	:= Axis_Halt.ErrorID;
	HaltDone 		:= Axis_Halt.Done;
	
	Axis_Move(	Execute	:= FALSE,
				Axis 	:= AxisRef);
				
	Axis_Halt(	Execute	:= FALSE,
				Axis 	:= AxisRef);
END_IF

// =========================================================
END_METHOD

METHOD Home
VAR_INPUT
	//Back_Start 				: BOOL;
	//Velocity_Home	:LREAL;
	//Axis_Current_Turque 	: INT;
	Drive_Home				: BOOL;
END_VAR

VAR
	//HomeSet					: BOOL;
	BackDone				: BOOL;					// 电机退回到顶点位，该标志位使能
END_VAR
// =======================找零程序==========================
// 找零程序过程为：先让丝杠回退，到达机械限位后停止,并用程序将该位置置为零位

//======================丝杠回退========================
Jog_Backward(Drive_Jog_Backward:= (Drive_Home AND (NOT BackDone)));
Jog_Velocity := Velocity_Home;
HomeDone := Axis_MoveAbsolute.Done;					// 找零结束的标志为丝杠伸长到制定距离
	
IF NOT Axis_Home.Error THEN
	IF ABS(Axis_Current_Turque) > Axis_Max_Turque AND NOT BackDone THEN
		//Drive_Home :=0;
		Jog_Backward(Drive_Jog_Backward:= 0);
		Delay(IN:= NOT Delay.Q, PT:=T#200MS, Q=> , ET=> );
		Axis_Home( 	Axis:= AxisRef, 
					Execute:= Delay.Q, 
					Position:= 0, 
					HomingMode:= MC_Direct);
		BackDone := Axis_Home.Done;				
	END_IF
	IF BackDone AND Drive_Home THEN
		Move_Absolute(Drive_Move_Absolute:= TRUE, Absolute_Position:= Home_Position );
		IF Axis_MoveAbsolute.Done THEN
			BackDone := FALSE;
			Drive_Home	:= FALSE;
		END_IF
	END_IF
END_IF

(*IF HomeSet THEN
	Jog_Backward(Drive_Jog_Backward:= 0,  Axis_Current_Turque:= Axis_Current_Turque);
	HomeDone := 1;
END_IF*)

IF Axis_Home.Error OR Axis_Home.CommandAborted OR ABS(Axis_Current_Turque) < Axis_Max_Turque THEN
	IF Axis_Jog.Error THEN
		Axis_Error		:= TRUE;
		Axis_ErrorID 	:= Axis_Home.ErrorID;
	END_IF
	Axis_Home( 	Axis:= AxisRef, 
				Execute:= FALSE);
END_IF

// =========================================================
END_METHOD

PROPERTY Home_Absolute_Position : LREAL
GET
Home_Absolute_Position := Home_Position;
END_GET
SET
Home_Position := Home_Absolute_Position;
END_SET
END_PROPERTY

METHOD Home_Sensor
VAR_INPUT
	Drive_Home				: BOOL;			// 调零使能信号
	Home_Switch				: BOOL;			// 零位调零传感器信号
	//MaxPosition_Swicth		: BOOL;
END_VAR

VAR
	//HomeSet				: BOOL;
	BackDone				: BOOL;					// 电机退回到顶点位，该标志位使能
END_VAR
// =======================找零程序==========================
// 找零程序过程为：先让丝杠回退，当传感器检测到金属表面并反馈信号后, 程序将该位置置为零位

//======================丝杠回退========================
Jog_Backward(Drive_Jog_Backward:= Drive_Home);
Jog_Velocity := Velocity_Home;
HomeDone := Axis_MoveAbsolute.Done;					// 回到零点的标志为丝杠伸长到制定距离
	
IF NOT Axis_Home.Error THEN
	IF Home_Switch AND NOT HomeDone THEN
		Drive_Home :=0;
		Jog_Backward(Drive_Jog_Backward:= Drive_Home);
		Delay(IN:= NOT Delay.Q, PT:=T#200MS, Q=> , ET=> );
		Axis_Home( 	Axis:= AxisRef, 
					Execute:= Delay.Q,
					Position:= 0, 
					HomingMode:= MC_Direct);
		BackDone := Axis_Home.Done;
	END_IF
	IF BackDone THEN
		Move_Absolute(Drive_Move_Absolute:= TRUE, Absolute_Position:= 20);
		IF Axis_MoveAbsolute.Done THEN
			BackDone := FALSE;
		END_IF
	END_IF
END_IF

(*IF HomeSet THEN
	Jog_Backward(Drive_Jog_Backward:= 0,  Axis_Current_Turque:= Axis_Current_Turque);
	HomeDone := 1;
END_IF*)

IF Axis_Home.Error OR Axis_Home.CommandAborted OR ABS(Axis_Current_Turque) < Axis_Max_Turque THEN
	IF Axis_Jog.Error THEN
		Axis_Error		:= TRUE;
		Axis_ErrorID 	:= Axis_Home.ErrorID;
	END_IF
	Axis_Home( 	Axis:= AxisRef, 
				Execute:= FALSE);
END_IF

// =========================================================
END_METHOD

PROPERTY Home_Velocity : LREAL
GET
Home_Velocity := Velocity_Home;
END_GET
SET
Velocity_Home := Home_Velocity;
END_SET
END_PROPERTY

METHOD Jog_Backward
VAR_INPUT
	Drive_Jog_Backward	: BOOL;				//点动后退使能信号
	//Velocity_Jog		: LREAL;			//点动速度
	//Axis_Current_Turque : INT;				//边界条件：丝杠位置到达两端卡死
END_VAR
// =======================点动后退==========================
// 点动后退用在找零中的位置移动

IF NOT Axis_Jog.Error THEN
	Axis_Jog( 	Axis:= AxisRef, 
				JogForward:= 0, 
				JogBackwards:= Drive_Jog_Backward, 
				Mode:= MC_JOGMODE_CONTINOUS, 
				Velocity:= Velocity_Jog);
END_IF

IF Axis_Jog.Error OR Axis_Jog.CommandAborted OR ABS(Axis_Current_Turque) > Axis_Max_Turque THEN
	IF Axis_Jog.Error THEN
		Axis_Error		:= TRUE;
		Axis_ErrorID 	:= Axis_Jog.ErrorID;
	END_IF
	
	Axis_Jog(	JogForward:= 0, 
				JogBackwards:= 0, 
				Axis := AxisRef);
END_IF

(*IF ABS(Axis_Current_Turque) <1000 AND JogDone =1 THEN
	Axis_Jog(	JogForward:= 0, 
				JogBackwards:= 0, 
				Axis := AxisRef);
	JogDone :=0;
END_IF*)
				
// =========================================================
END_METHOD

METHOD Jog_Forward : BOOL
VAR_INPUT
	Drive_Jog_Forward	: BOOL;				//点动前进使能信号
	//Velocity_Jog		: LREAL;			//点动速度
	//Axis_Current_Turque : INT;				//边界条件：丝杠位置到达两端卡死
END_VAR
// =======================点动前进==========================


IF NOT Axis_Jog.Error THEN
	Axis_Jog( 	Axis:= AxisRef, 
				JogForward:= Drive_Jog_Forward, 
				JogBackwards:= 0, 
				Mode:= MC_JOGMODE_CONTINOUS, 
				Velocity:= Velocity_Jog);
END_IF

IF Axis_Jog.Error OR Axis_Jog.CommandAborted OR ABS(Axis_Current_Turque) > Axis_Max_Turque THEN
	IF Axis_Jog.Error THEN
		Axis_Error		:= TRUE;
		Axis_ErrorID 	:= Axis_Jog.ErrorID;
	END_IF
	
	Axis_Jog(	JogForward:= 0, 
				JogBackwards:= 0, 
				Axis := AxisRef);
END_IF

(*IF ABS(Axis_Current_Turque) <1000 AND JogDone =1 THEN
	Axis_Jog(	JogForward:= 0, 
				JogBackwards:= 0, 
				Axis := AxisRef);
	JogDone :=0;
END_IF*)
				
// =========================================================
END_METHOD

// =======================读写点动程序中的速度值==========================

PROPERTY Jog_Velocity : LREAL
GET
Jog_Velocity := Velocity_Jog;
END_GET
SET
Velocity_Jog := Jog_Velocity;
END_SET
END_PROPERTY

PROPERTY Max_Turque_Value : INT
SET
Axis_Max_Turque := Max_Turque_Value;
END_SET
END_PROPERTY

METHOD Move_Absolute
VAR_INPUT
	Drive_Move_Absolute : BOOL;				// 运动使能信号
	Absolute_Position	: LREAL;			// 绝对运动位置
	//Move_Velocity		: LREAL;			// 运动速度
	//Axis_Current_Turque : INT;			// 边界条件：丝杠位置到达两端卡死
END_VAR
// =======================绝对运动==========================

IF NOT Axis_MoveAbsolute.Error THEN
	Axis_MoveAbsolute(	Axis:= AxisRef, 
						Execute:= Drive_Move_Absolute, 
						Position:= Absolute_Position, 
						Velocity:= Velocity_Absolute, 
						BufferMode:= MC_Aborting );
	MoveAbsoluteDone := Axis_MoveAbsolute.Done;			// 运动到指定位置后置位
END_IF

IF Axis_MoveAbsolute.Error OR Axis_MoveAbsolute.CommandAborted OR ABS(Axis_Current_Turque) > Axis_Max_Turque THEN
	IF Axis_MoveAbsolute.Error THEN
		Axis_Error		:= TRUE;
		Axis_ErrorID 	:= Axis_MoveAbsolute.ErrorID;
	END_IF
	
	Axis_MoveAbsolute(	Axis:= AxisRef, 
						Execute:= 0, 
						BufferMode:= MC_Aborting);
END_IF

// =========================================================
END_METHOD

// =======================读写绝对运动程序中的速度值==========================

PROPERTY Move_Absolute_Velocity : LREAL
GET
Move_Absolute_Velocity := Velocity_Absolute;
END_GET
SET
Velocity_Absolute := Move_Absolute_Velocity;
END_SET
END_PROPERTY

METHOD Move_Backward
VAR_INPUT
	Move_Backward_Start : BOOL;					//匀速后退使能信号
	//Axis_Current_Turque : INT;					//边界条件：丝杠位置到达两端卡死
END_VAR
// =======================匀速后退==========================

// Not error
IF NOT Axis_Move.Error THEN
	Axis_Move(	Execute 	:= Move_Backward_Start,
				Velocity 	:= Velocity_Move,
				Direction 	:= MC_Negative_Direction,
				Axis 		:= AxisRef );
END_IF

// Error / Command aborted
IF Axis_Move.Error OR Axis_Move.CommandAborted OR ABS(Axis_Current_Turque) > Axis_Max_Turque THEN
	IF Axis_Move.Error THEN
		Axis_Error		:= TRUE;
		Axis_ErrorID 	:= Axis_Move.ErrorID;
	END_IF
	
	Axis_Move(	Execute	:= FALSE,
				Axis 	:= AxisRef);
END_IF

// =========================================================
END_METHOD

METHOD Move_Fordward
VAR_INPUT
	Move_Forward_Start : BOOL;					//匀速前进使能信号
	//Axis_Current_Turque : INT;					//边界条件：丝杠位置到达两端卡死
END_VAR
// =======================匀速前进==========================

// Not error
IF NOT Axis_Move.Error THEN
	Axis_Move(	Execute 	:= Move_Forward_Start,
				Velocity 	:= Velocity_Move,
				Direction 	:= MC_Positive_Direction,
				Axis 		:= AxisRef );
END_IF

// Error / Command aborted
IF Axis_Move.Error OR Axis_Move.CommandAborted OR ABS(Axis_Current_Turque) > Axis_Max_Turque THEN
	IF Axis_Move.Error THEN
		Axis_Error		:= TRUE;
		Axis_ErrorID 	:= Axis_Move.ErrorID;
	END_IF
	
	Axis_Move(	Execute	:= FALSE,
				Axis 	:= AxisRef);
END_IF

// =========================================================
END_METHOD

METHOD Move_Relative
VAR_INPUT
	Drive_Move_Relative		: BOOL;				// 运动使能信号
	Relative_Position		: LREAL;			// 相对运动位置
	//Move_Velocity			: LREAL;			// 运动速度
	//Axis_Current_Turque 	: INT;				// 边界条件：丝杠位置到达两端卡死
END_VAR
// =======================相对运动==========================

IF NOT Axis_MoveRelative.Error THEN
	Axis_MoveRelative(	Axis:= AxisRef, 
						Execute:= Drive_Move_Relative, 
						Distance:= Relative_Position, 
						Velocity:= Velocity_Relative, 
						BufferMode:= MC_Aborting );
END_IF

IF Axis_MoveRelative.Error OR Axis_MoveRelative.CommandAborted OR ABS(Axis_Current_Turque) > Axis_Max_Turque THEN
	IF Axis_MoveRelative.Error THEN
		Axis_Error		:= TRUE;
		Axis_ErrorID 	:= Axis_MoveRelative.ErrorID;
	END_IF
	
	Axis_MoveRelative(	Axis:= AxisRef, 
						Execute:= 0, 
						BufferMode:= MC_Aborting);
END_IF

// =========================================================
END_METHOD

// =======================读写相对运动程序中的速度值==========================

PROPERTY Move_Relative_Velocity : LREAL
GET
Move_Relative_Velocity := Velocity_Relative;
END_GET
SET
Velocity_Relative := Move_Relative_Velocity;
END_SET
END_PROPERTY

PROPERTY Move_Velocity : LREAL
GET
Move_Velocity := Velocity_Move;
END_GET
SET
Velocity_Move :=Move_Velocity :=10;
END_SET
END_PROPERTY

METHOD Power
VAR_INPUT
	Axis_Enable : BOOL;
END_VAR
// =======================上电程序==========================

Axis_Power(	Enable 			:= Axis_Enable, 
			Enable_Positive	:= Axis_Enable, 
			Enable_Negative	:= Axis_Enable, 
			Override		:= fOverride,
			Axis			:= AxisRef,
			Status			=> Power_StatusEnable);
			
IF Axis_Power.Error THEN
	Axis_Error		:= TRUE;
	Axis_ErrorID 	:= Axis_Power.ErrorID;
END_IF

AxisRef.ReadStatus();

Axis_Moves := AxisRef.Status.Moving;

// ==========================================================
END_METHOD

METHOD Reset
VAR_INPUT
	Drive_Reset		: BOOL;					// Request reset
END_VAR
// =====================驱动重置程序==========================

IF NOT Drive_Reset THEN
	ResetDone 	:= FALSE;
END_IF

// Trigger(触发器)
TriggerReset(CLK := Drive_Reset);

IF TriggerReset.Q THEN
	HaltDone 	:= FALSE;
	
	Axis_Reset(Execute := TRUE, Axis := AxisRef);
ELSE
	Axis_Reset(Axis := AxisRef);
END_IF

